KUKA KRL program: MyProgram_219().src

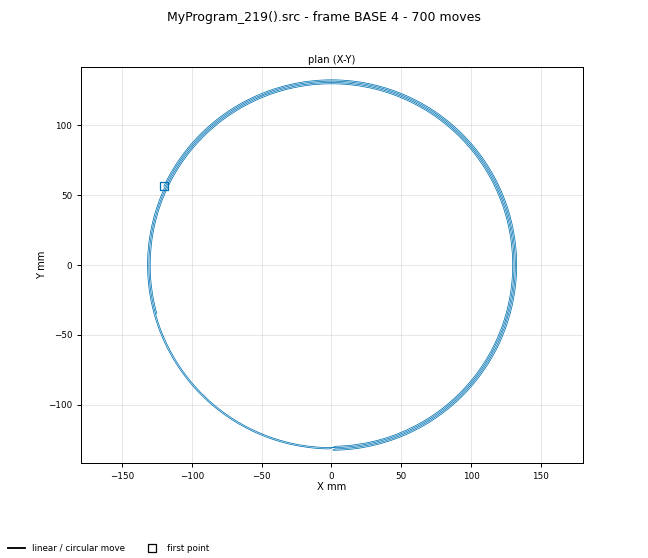
[picture p0: tool path of MyProgram_219().src in frame BASE 4, 700 of 700 moves have a stored position in this frame; points joined in program order, loops and branches not executed]
&ACCESS RVP
&REL 1
&PARAM TEMPLATE = C:\KRC\Roboter\Template\vorgabe
&PARAM EDITMASK = *
DEF MyProgram_219()
; ---- Setting reference (Base) ----
$BASE = BASE_DATA[4]

; --------------------------
; ---- Setting tool (TCP) ----
$TOOL = TOOL_DATA[3]
; --------------------------

$VEL.CP = VEL_APROX_PRINT
Startdeposition()
$VEL.CP = VEL_PRINT
LIN {X -120.0185,Y 56.4143,Z 153,A 151.3812,B 23.2874,C -1.2198,E1 23.1731,E2 655.6773} C_DIS
LIN {X -118.5604,Y 59.4176,Z 153,A 149.9276,B 23.2872,C -1.2236,E1 23.1749,E2 657.1297} C_DIS
LIN {X -117.0207,Y 62.3953,Z 153,A 148.4681,B 23.287,C -1.2274,E1 23.1767,E2 658.5879} C_DIS
LIN {X -115.456,Y 65.2445,Z 153,A 146.9748,B 23.287,C -1.2276,E1 23.1788,E2 660.0893} C_DIS
LIN {X -113.2613,Y 68.9846,Z 153,A 145.0626,B 23.2868,C -1.2313,E1 23.1815,E2 662.0028} C_DIS
LIN {X -110.999,Y 72.5688,Z 153,A 143.3218,B 23.2864,C -1.2405,E1 23.1841,E2 663.7297} C_DIS
LIN {X -108.7297,Y 75.9258,Z 153,A 141.4715,B 23.2864,C -1.2409,E1 23.1871,E2 665.5888} C_DIS
LIN {X -106.1126,Y 79.5432,Z 153,A 139.5664,B 23.286,C -1.2472,E1 23.1902,E2 667.4879} C_DIS
LIN {X -103.5175,Y 82.8922,Z 153,A 137.6938,B 23.2859,C -1.2502,E1 23.1934,E2 669.3624} C_DIS
LIN {X -100.7633,Y 86.2193,Z 153,A 135.8973,B 23.2855,C -1.2582,E1 23.1966,E2 671.1476} C_DIS
LIN {X -98.5031,Y 88.7927,Z 153,A 134.4081,B 23.2853,C -1.2615,E1 23.1994,E2 672.6355} C_DIS
LIN {X -96.2052,Y 91.2772,Z 153,A 132.8552,B 23.2853,C -1.2611,E1 23.2024,E2 674.1968} C_DIS
LIN {X -93.1648,Y 94.3786,Z 153,A 131.0513,B 23.2849,C -1.2689,E1 23.2059,E2 675.9891} C_DIS
LIN {X -90.6941,Y 96.7553,Z 153,A 129.562,B 23.2848,C -1.2721,E1 23.2089,E2 677.4771} C_DIS
LIN {X -88.1572,Y 99.0723,Z 153,A 128.0728,B 23.2846,C -1.2753,E1 23.212,E2 678.9646} C_DIS
LIN {X -85.3531,Y 101.4973,Z 153,A 126.3626,B 23.2846,C -1.274,E1 23.2157,E2 680.6852} C_DIS
LIN {X -82.2555,Y 104.0242,Z 153,A 124.7251,B 23.2843,C -1.2818,E1 23.2192,E2 682.3096} C_DIS
LIN {X -79.5467,Y 106.11,Z 153,A 123.2418,B 23.2841,C -1.2846,E1 23.2225,E2 683.7914} C_DIS
LIN {X -76.3743,Y 108.415,Z 153,A 121.4898,B 23.2841,C -1.2855,E1 23.2265,E2 685.5479} C_DIS
LIN {X -73.2819,Y 110.5295,Z 153,A 119.9361,B 23.2838,C -1.2916,E1 23.2301,E2 687.0917} C_DIS
LIN {X -70.2231,Y 112.497,Z 153,A 118.2317,B 23.2839,C -1.2885,E1 23.2341,E2 688.8097} C_DIS
LIN {X -66.2198,Y 114.8992,Z 153,A 116.2269,B 23.2837,C -1.2927,E1 23.2389,E2 690.8105} C_DIS
LIN {X -62.3991,Y 117.0186,Z 153,A 114.4206,B 23.2833,C -1.2996,E1 23.2433,E2 692.6047} C_DIS
LIN {X -59.4253,Y 118.5564,Z 153,A 112.9705,B 23.2833,C -1.3018,E1 23.2469,E2 694.0535} C_DIS
LIN {X -56.8721,Y 119.7998,Z 153,A 111.7391,B 23.2831,C -1.3036,E1 23.25,E2 695.2838} C_DIS
LIN {X -53.3965,Y 121.3912,Z 153,A 110.0849,B 23.2831,C -1.3059,E1 23.2542,E2 696.9365} C_DIS
LIN {X -50.3517,Y 122.6854,Z 153,A 108.6524,B 23.2829,C -1.3078,E1 23.2579,E2 698.3678} C_DIS
LIN {X -47.2831,Y 123.9004,Z 153,A 107.2236,B 23.2829,C -1.3096,E1 23.2616,E2 699.7954} C_DIS
LIN {X -44.4516,Y 124.9428,Z 153,A 105.9301,B 23.2827,C -1.3117,E1 23.265,E2 701.0862} C_DIS
LIN {X -41.1344,Y 126.0752,Z 153,A 104.4014,B 23.2827,C -1.3128,E1 23.2691,E2 702.6152} C_DIS
LIN {X -38.0368,Y 127.0441,Z 153,A 102.9974,B 23.2826,C -1.3143,E1 23.2728,E2 704.018} C_DIS
LIN {X -34.9435,Y 127.9295,Z 153,A 101.606,B 23.2825,C -1.3157,E1 23.2766,E2 705.4082} C_DIS
LIN {X -31.8497,Y 128.7346,Z 153,A 100.2237,B 23.2825,C -1.317,E1 23.2803,E2 706.7893} C_DIS
LIN {X -28.7581,Y 129.4603,Z 153,A 98.8511,B 23.2824,C -1.3182,E1 23.284,E2 708.1608} C_DIS
LIN {X -26.1134,Y 130.0177,Z 153,A 97.6447,B 23.2824,C -1.3174,E1 23.2873,E2 709.3708} C_DIS
LIN {X -22.593,Y 130.6773,Z 153,A 96.0716,B 23.2824,C -1.3174,E1 23.2917,E2 710.9459} C_DIS
LIN {X -18.9352,Y 131.2551,Z 153,A 94.4964,B 23.2823,C -1.3196,E1 23.296,E2 712.5168} C_DIS
LIN {X -15.475,Y 131.708,Z 153,A 92.9768,B 23.2823,C -1.3199,E1 23.3002,E2 714.0368} C_DIS
LIN {X -11.9161,Y 132.0796,Z 153,A 91.4838,B 23.2821,C -1.3231,E1 23.3043,E2 715.5225} C_DIS
LIN {X -8.9319,Y 132.3147,Z 153,A 90.1919,B 23.2821,C -1.3238,E1 23.3079,E2 716.8134} C_DIS
LIN {X -5.3392,Y 132.5065,Z 153,A 88.5959,B 23.2821,C -1.3223,E1 23.3124,E2 718.4133} C_DIS
LIN {X -1.9248,Y 132.6003,Z 153,A 87.1244,B 23.2821,C -1.3229,E1 23.3165,E2 719.8836} C_DIS
LIN {X 2.9359,Y 132.5835,Z 153,A 84.8957,B 23.2824,C -1.3171,E1 23.3228,E2 722.1267} C_DIS
LIN {X 6.6279,Y 132.4482,Z 153,A 83.4443,B 23.282,C -1.3241,E1 23.3268,E2 723.5601} C_DIS
LIN {X 9.8143,Y 132.2503,Z 153,A 82.0646,B 23.282,C -1.324,E1 23.3306,E2 724.9392} C_DIS
LIN {X 13.086,Y 131.9673,Z 153,A 80.635,B 23.282,C -1.3233,E1 23.3346,E2 726.3697} C_DIS
LIN {X 16.4617,Y 131.5903,Z 153,A 79.1907,B 23.282,C -1.3241,E1 23.3386,E2 727.8108} C_DIS
LIN {X 20.6084,Y 131.0031,Z 153,A 77.3967,B 23.282,C -1.3243,E1 23.3435,E2 729.6025} C_DIS
LIN {X 23.6048,Y 130.4963,Z 153,A 76.0345,B 23.2822,C -1.3215,E1 23.3473,E2 730.9703} C_DIS
LIN {X 26.916,Y 129.8544,Z 153,A 74.5879,B 23.2822,C -1.3213,E1 23.3513,E2 732.4155} C_DIS
LIN {X 30.2955,Y 129.1092,Z 153,A 73.1112,B 23.2822,C -1.3213,E1 23.3553,E2 733.8899} C_DIS
LIN {X 33.027,Y 128.4359,Z 153,A 71.8933,B 23.2822,C -1.3205,E1 23.3586,E2 735.1079} C_DIS
LIN {X 36.4824,Y 127.4991,Z 153,A 70.349,B 23.2822,C -1.3195,E1 23.3627,E2 736.652} C_DIS
LIN {X 39.0613,Y 126.7306,Z 153,A 69.134,B 23.2825,C -1.3161,E1 23.366,E2 737.8732} C_DIS
LIN {X 42.669,Y 125.5642,Z 153,A 67.5494,B 23.2825,C -1.3173,E1 23.3702,E2 739.4515} C_DIS
LIN {X 45.3374,Y 124.6235,Z 153,A 66.2925,B 23.2825,C -1.3145,E1 23.3735,E2 740.7126} C_DIS
LIN {X 48.8073,Y 123.3079,Z 153,A 64.7278,B 23.2825,C -1.3147,E1 23.3776,E2 742.2731} C_DIS
LIN {X 51.3866,Y 122.2532,Z 153,A 63.4941,B 23.2827,C -1.312,E1 23.3807,E2 743.5105} C_DIS
LIN {X 54.6118,Y 120.8476,Z 153,A 61.9862,B 23.2827,C -1.3109,E1 23.3846,E2 745.0173} C_DIS
LIN {X 57.9189,Y 119.2997,Z 153,A 60.4317,B 23.2827,C -1.31,E1 23.3885,E2 746.5696} C_DIS
LIN {X 60.9098,Y 117.8007,Z 153,A 58.9892,B 23.2829,C -1.3083,E1 23.3921,E2 748.0122} C_DIS
LIN {X 63.403,Y 116.477,Z 153,A 57.6835,B 23.2832,C -1.3024,E1 23.3953,E2 749.3287} C_DIS
LIN {X 67.2041,Y 114.3261,Z 153,A 55.8328,B 23.2832,C -1.3014,E1 23.3998,E2 751.1759} C_DIS
LIN {X 70.7142,Y 112.1889,Z 153,A 54.0427,B 23.2834,C -1.2979,E1 23.4041,E2 752.9686} C_DIS
LIN {X 74.3709,Y 109.7989,Z 153,A 52.1811,B 23.2835,C -1.2961,E1 23.4084,E2 754.8281} C_DIS
LIN {X 77.7327,Y 107.4452,Z 153,A 50.3815,B 23.2838,C -1.2917,E1 23.4125,E2 756.632} C_DIS
LIN {X 81.1809,Y 104.8642,Z 153,A 48.5353,B 23.2838,C -1.2891,E1 23.4166,E2 758.4776} C_DIS
LIN {X 84.2506,Y 102.4151,Z 153,A 46.9275,B 23.2838,C -1.2902,E1 23.4201,E2 760.0759} C_DIS
LIN {X 87.0607,Y 100.0365,Z 153,A 45.2407,B 23.2842,C -1.2823,E1 23.4237,E2 761.7756} C_DIS
LIN {X 90.0629,Y 97.3431,Z 153,A 43.608,B 23.2842,C -1.2842,E1 23.427,E2 763.3963} C_DIS
LIN {X 92.9608,Y 94.5787,Z 153,A 41.865,B 23.2844,C -1.2799,E1 23.4305,E2 765.1423} C_DIS
LIN {X 95.7389,Y 91.7656,Z 153,A 40.0792,B 23.2848,C -1.2723,E1 23.434,E2 766.939} C_DIS
LIN {X 98.4971,Y 88.7993,Z 153,A 38.3818,B 23.2848,C -1.2709,E1 23.4372,E2 768.6317} C_DIS
LIN {X 101.3154,Y 85.5698,Z 153,A 36.6033,B 23.2848,C -1.2703,E1 23.4404,E2 770.4031} C_DIS
LIN {X 103.4942,Y 82.9214,Z 153,A 35.136,B 23.285,C -1.2674,E1 23.443,E2 771.8702} C_DIS
LIN {X 105.8539,Y 79.8861,Z 153,A 33.4134,B 23.2854,C -1.2602,E1 23.446,E2 773.602} C_DIS
LIN {X 108.1241,Y 76.7866,Z 153,A 31.8291,B 23.2854,C -1.2598,E1 23.4485,E2 775.1791} C_DIS
LIN {X 110.3638,Y 73.5301,Z 153,A 30.0564,B 23.2858,C -1.2522,E1 23.4513,E2 776.9616} C_DIS
LIN {X 112.7423,Y 69.829,Z 153,A 28.1496,B 23.2861,C -1.2468,E1 23.4542,E2 778.8715} C_DIS
LIN {X 114.9822,Y 66.0764,Z 153,A 26.3687,B 23.2861,C -1.2471,E1 23.4567,E2 780.6416} C_DIS
LIN {X 116.7068,Y 62.9795,Z 153,A 24.731,B 23.2865,C -1.2375,E1 23.4589,E2 782.2942} C_DIS
LIN {X 118.5564,Y 59.4253,Z 153,A 23.1289,B 23.2865,C -1.2392,E1 23.4609,E2 783.8829} C_DIS
LIN {X 120.0148,Y 56.4221,Z 153,A 21.6972,B 23.2866,C -1.2356,E1 23.4626,E2 785.3153} C_DIS
LIN {X 121.2676,Y 53.6728,Z 153,A 20.4109,B 23.2868,C -1.2329,E1 23.4641,E2 786.601} C_DIS
LIN {X 122.5698,Y 50.6284,Z 153,A 18.9867,B 23.287,C -1.229,E1 23.4657,E2 788.0264} C_DIS
LIN {X 123.8752,Y 47.3479,Z 153,A 17.4806,B 23.2871,C -1.2255,E1 23.4672,E2 789.5324} C_DIS
LIN {X 124.8207,Y 44.7903,Z 153,A 16.2864,B 23.2874,C -1.2212,E1 23.4683,E2 790.7302} C_DIS
LIN {X 126.052,Y 41.204,Z 153,A 14.6728,B 23.2875,C -1.2174,E1 23.4698,E2 792.3434} C_DIS
LIN {X 127.0441,Y 38.0368,Z 153,A 13.2519,B 23.2877,C -1.2137,E1 23.4709,E2 793.7648} C_DIS
LIN {X 127.9112,Y 35.009,Z 153,A 11.9126,B 23.2879,C -1.2106,E1 23.4719,E2 795.1035} C_DIS
LIN {X 128.7346,Y 31.8497,Z 153,A 10.5038,B 23.2881,C -1.2063,E1 23.4729,E2 796.5144} C_DIS
LIN {X 129.4603,Y 28.7581,Z 153,A 9.1435,B 23.2883,C -1.2026,E1 23.4738,E2 797.8754} C_DIS
LIN {X 130.1059,Y 25.6797,Z 153,A 7.7968,B 23.2884,C -1.199,E1 23.4745,E2 799.2228} C_DIS
LIN {X 130.5831,Y 23.1195,Z 153,A 6.7047,B 23.2885,C -1.1972,E1 23.4751,E2 800.3126} C_DIS
LIN {X 131.0734,Y 20.1545,Z 153,A 5.3619,B 23.2888,C -1.1908,E1 23.4757,E2 801.663} C_DIS
LIN {X 131.5883,Y 16.4774,Z 153,A 3.8042,B 23.289,C -1.188,E1 23.4762,E2 803.2177} C_DIS
LIN {X 131.9334,Y 13.4374,Z 153,A 2.4944,B 23.2891,C -1.1844,E1 23.4766,E2 804.5282} C_DIS
LIN {X 132.2472,Y 9.8566,Z 153,A 0.9066,B 23.2895,C -1.1776,E1 23.477,E2 806.1228} C_DIS
LIN {X 132.4544,Y 6.5035,Z 153,A -0.5469,B 23.2897,C -1.1728,E1 23.4772,E2 807.5791} C_DIS
LIN {X 132.5999,Y 1.951,Z 153,A -2.4995,B 23.29,C -1.1672,E1 23.4774,E2 809.5332} C_DIS
LIN {X 132.6105,Y -0.9415,Z 153,A -3.7215,B 23.29,C -1.1645,E1 23.4774,E2 810.7539} C_DIS
LIN {X 132.5171,Y -5.0689,Z 153,A -5.4928,B 23.2903,C -1.1594,E1 23.4772,E2 812.5269} C_DIS
LIN {X 132.3401,Y -8.5247,Z 153,A -6.9651,B 23.2905,C -1.1557,E1 23.477,E2 813.999} C_DIS
LIN {X 132.0802,Y -11.9083,Z 153,A -8.3941,B 23.2906,C -1.1528,E1 23.4766,E2 815.4262} C_DIS
LIN {X 131.6676,Y -15.8141,Z 153,A -10.1033,B 23.2909,C -1.1466,E1 23.4761,E2 817.1398} C_DIS
LIN {X 131.2563,Y -18.9271,Z 153,A -11.466,B 23.2911,C -1.1419,E1 23.4756,E2 818.5057} C_DIS
LIN {X 130.6787,Y -22.5851,Z 153,A -13.0213,B 23.2913,C -1.139,E1 23.4749,E2 820.0585} C_DIS
LIN {X 130.1811,Y -25.2871,Z 153,A -14.2322,B 23.2915,C -1.134,E1 23.4742,E2 821.2744} C_DIS
LIN {X 129.4621,Y -28.7502,Z 153,A -15.7214,B 23.2917,C -1.131,E1 23.4734,E2 822.7616} C_DIS
LIN {X 128.5056,Y -32.7522,Z 153,A -17.5015,B 23.2919,C -1.1252,E1 23.4722,E2 824.5451} C_DIS
LIN {X 127.6253,Y -36.0315,Z 153,A -18.9893,B 23.2922,C -1.1195,E1 23.4711,E2 826.0382} C_DIS
LIN {X 126.5736,Y -39.5742,Z 153,A -20.5353,B 23.2922,C -1.117,E1 23.4698,E2 827.5809} C_DIS
LIN {X 125.6993,Y -42.2632,Z 153,A -21.7708,B 23.2925,C -1.1124,E1 23.4687,E2 828.8203} C_DIS
LIN {X 124.4755,Y -45.7477,Z 153,A -23.3361,B 23.2927,C -1.109,E1 23.4673,E2 830.3848} C_DIS
LIN {X 123.3079,Y -48.8073,Z 153,A -24.741,B 23.2928,C -1.1051,E1 23.4659,E2 831.791} C_DIS
LIN {X 122.2841,Y -51.3126,Z 153,A -25.9212,B 23.293,C -1.101,E1 23.4646,E2 832.9745} C_DIS
LIN {X 120.9147,Y -54.4616,Z 153,A -27.371,B 23.2931,C -1.0981,E1 23.463,E2 834.4229} C_DIS
LIN {X 119.5106,Y -57.4773,Z 153,A -28.828,B 23.2934,C -1.0928,E1 23.4612,E2 835.8849} C_DIS
LIN {X 117.8007,Y -60.9098,Z 153,A -30.4567,B 23.2935,C -1.0892,E1 23.4592,E2 837.5132} C_DIS
LIN {X 116.3772,Y -63.586,Z 153,A -31.8054,B 23.2938,C -1.0833,E1 23.4574,E2 838.8689} C_DIS
LIN {X 114.2709,Y -67.298,Z 153,A -33.6824,B 23.2941,C -1.0763,E1 23.4547,E2 840.7533} C_DIS
LIN {X 111.921,Y -71.1386,Z 153,A -35.5264,B 23.2941,C -1.0758,E1 23.452,E2 842.5883} C_DIS
LIN {X 109.8274,Y -74.3288,Z 153,A -37.232,B 23.2944,C -1.0683,E1 23.4494,E2 844.3037} C_DIS
LIN {X 107.6309,Y -77.4765,Z 153,A -38.8145,B 23.2944,C -1.0675,E1 23.4468,E2 845.8797} C_DIS
LIN {X 105.5981,Y -80.225,Z 153,A -40.2823,B 23.2946,C -1.064,E1 23.4444,E2 847.3489} C_DIS
LIN {X 103.4942,Y -82.9214,Z 153,A -41.835,B 23.295,C -1.0562,E1 23.4416,E2 848.9134} C_DIS
LIN {X 100.7633,Y -86.2193,Z 153,A -43.5915,B 23.295,C -1.0561,E1 23.4385,E2 850.6615} C_DIS
LIN {X 98.5031,Y -88.7927,Z 153,A -45.0636,B 23.2951,C -1.0527,E1 23.4358,E2 852.135} C_DIS
LIN {X 96.1695,Y -91.315,Z 153,A -46.5193,B 23.2952,C -1.0504,E1 23.433,E2 853.5895} C_DIS
LIN {X 93.7768,Y -93.7705,Z 153,A -48.1152,B 23.2956,C -1.0409,E1 23.4298,E2 855.202} C_DIS
LIN {X 90.6941,Y -96.7553,Z 153,A -49.8566,B 23.2956,C -1.0422,E1 23.4263,E2 856.9323} C_DIS
LIN {X 88.1572,Y -99.0723,Z 153,A -51.3324,B 23.2956,C -1.0391,E1 23.4233,E2 858.4094} C_DIS
LIN {X 85.5698,Y -101.3154,Z 153,A -52.7981,B 23.2958,C -1.0364,E1 23.4202,E2 859.8757} C_DIS
LIN {X 82.6822,Y -103.6846,Z 153,A -54.5007,B 23.2961,C -1.0284,E1 23.4164,E2 861.5916} C_DIS
LIN {X 79.0894,Y -106.4505,Z 153,A -56.3994,B 23.2961,C -1.0272,E1 23.4122,E2 863.4857} C_DIS
LIN {X 75.5577,Y -108.9858,Z 153,A -58.3154,B 23.2964,C -1.0215,E1 23.4078,E2 865.4091} C_DIS
LIN {X 71.8604,Y -111.4589,Z 153,A -60.14,B 23.2964,C -1.0226,E1 23.4036,E2 867.2244} C_DIS
LIN {X 68.9846,Y -113.2613,Z 153,A -61.5988,B 23.2964,C -1.0202,E1 23.4001,E2 868.6843} C_DIS
LIN {X 66.0764,Y -114.9822,Z 153,A -63.0515,B 23.2966,C -1.0179,E1 23.3966,E2 870.1379} C_DIS
LIN {X 62.8825,Y -116.7589,Z 153,A -64.7151,B 23.2969,C -1.0109,E1 23.3925,E2 871.8139} C_DIS
LIN {X 59.4253,Y -118.5564,Z 153,A -66.2983,B 23.2968,C -1.0131,E1 23.3886,E2 873.3869} C_DIS
LIN {X 56.9163,Y -119.7787,Z 153,A -67.494,B 23.2968,C -1.0117,E1 23.3856,E2 874.5827} C_DIS
LIN {X 53.8486,Y -121.1889,Z 153,A -68.9478,B 23.2969,C -1.0097,E1 23.3819,E2 876.0377} C_DIS
LIN {X 50.6868,Y -122.5454,Z 153,A -70.4194,B 23.2969,C -1.0082,E1 23.3781,E2 877.5092} C_DIS
LIN {X 47.2831,Y -123.9004,Z 153,A -72.0079,B 23.2971,C -1.0057,E1 23.374,E2 879.1002} C_DIS
LIN {X 44.707,Y -124.8507,Z 153,A -73.2383,B 23.2972,C -1.002,E1 23.3707,E2 880.3372} C_DIS
LIN {X 41.1344,Y -126.0752,Z 153,A -74.8143,B 23.2972,C -1.0027,E1 23.3666,E2 881.9081} C_DIS
LIN {X 38.0368,Y -127.0441,Z 153,A -76.211,B 23.2972,C -1.0014,E1 23.3628,E2 883.3056} C_DIS
LIN {X 34.9435,Y -127.9295,Z 153,A -77.5957,B 23.2973,C -1.0001,E1 23.3591,E2 884.6909} C_DIS
LIN {X 32.039,Y -128.6866,Z 153,A -78.8599,B 23.2973,C -1.0004,E1 23.3557,E2 885.9522} C_DIS
LIN {X 29.315,Y -129.3331,Z 153,A -80.1109,B 23.2974,C -0.9972,E1 23.3523,E2 887.2094} C_DIS
LIN {X 25.6797,Y -130.1059,Z 153,A -81.6928,B 23.2974,C -0.997,E1 23.348,E2 888.7898} C_DIS
LIN {X 22.9082,Y -130.6209,Z 153,A -82.9272,B 23.2975,C -0.9952,E1 23.3446,E2 890.0272} C_DIS
LIN {X 18.9609,Y -131.2514,Z 153,A -84.6446,B 23.2975,C -0.9945,E1 23.3398,E2 891.7447} C_DIS
LIN {X 15.7554,Y -131.6746,Z 153,A -86.0399,B 23.2975,C -0.9937,E1 23.336,E2 893.1408} C_DIS
LIN {X 12.4799,Y -132.0255,Z 153,A -87.4629,B 23.2975,C -0.9929,E1 23.332,E2 894.5647} C_DIS
LIN {X 8.9114,Y -132.3162,Z 153,A -88.9797,B 23.2975,C -0.9937,E1 23.3278,E2 896.0789} C_DIS
LIN {X 3.8989,Y -132.5568,Z 153,A -91.2084,B 23.2977,C -0.99,E1 23.3215,E2 898.3162} C_DIS
LIN {X 0.9369,Y -132.6077,Z 153,A -92.0457,B 23.2969,C -1.0112,E1 23.3194,E2 899.0997} C_DIS
Enddeposition()
LIN {X 0.9369,Y -132.6077,Z 153,A -92.0457,B 23.2969,C -1.0112,E1 23.3194,E2 899.0997} C_DIS
Startdeposition()
$VEL.CP = VEL_PRINT
LIN {X 2.3502,Y -131.6529,Z 153,A -90.8514,B 22.2978,C -0.8695,E1 22.3183,E2 898.1516} C_DIS
LIN {X 6.558,Y -131.5103,Z 153,A -89.0359,B 22.2978,C -0.8694,E1 22.3233,E2 896.337} C_DIS
LIN {X 10.8155,Y -131.229,Z 153,A -87.1803,B 22.2978,C -0.8702,E1 22.3285,E2 894.4805} C_DIS
LIN {X 14.3146,Y -130.8934,Z 153,A -85.6847,B 22.2978,C -0.8694,E1 22.3326,E2 892.9879} C_DIS
LIN {X 18.2026,Y -130.4101,Z 153,A -83.7965,B 22.2974,C -0.8791,E1 22.3379,E2 891.076} C_DIS
LIN {X 22.0211,Y -129.8196,Z 153,A -82.2316,B 22.2976,C -0.8748,E1 22.3422,E2 889.5241} C_DIS
LIN {X 27.5629,Y -128.7565,Z 153,A -80.0882,B 22.298,C -0.8621,E1 22.348,E2 887.4171} C_DIS
LIN {X 29.4629,Y -128.335,Z 153,A -79.0109,B 22.2976,C -0.8738,E1 22.351,E2 886.3108} C_DIS
LIN {X 33.0947,Y -127.4487,Z 153,A -77.3837,B 22.2976,C -0.8754,E1 22.3554,E2 884.6822} C_DIS
LIN {X 38.7328,Y -125.8479,Z 153,A -74.7637,B 22.2973,C -0.8815,E1 22.3625,E2 882.0511} C_DIS
LIN {X 42.1515,Y -124.7456,Z 153,A -73.3003,B 22.2974,C -0.8787,E1 22.3663,E2 880.5985} C_DIS
LIN {X 45.6252,Y -123.5174,Z 153,A -71.4667,B 22.2969,C -0.8918,E1 22.3712,E2 878.7347} C_DIS
LIN {X 49.9299,Y -121.8418,Z 153,A -69.6991,B 22.2973,C -0.8829,E1 22.3757,E2 876.9949} C_DIS
LIN {X 52.3421,Y -120.8228,Z 153,A -68.5334,B 22.2972,C -0.8859,E1 22.3787,E2 875.8246} C_DIS
LIN {X 55.6372,Y -119.342,Z 153,A -66.9756,B 22.2971,C -0.8876,E1 22.3827,E2 874.2667} C_DIS
LIN {X 59.9235,Y -117.2478,Z 153,A -64.8252,B 22.2968,C -0.8945,E1 22.3881,E2 872.1047} C_DIS
LIN {X 63.7063,Y -115.2383,Z 153,A -62.9608,B 22.2968,C -0.8977,E1 22.3927,E2 870.2379} C_DIS
LIN {X 67.6763,Y -112.9529,Z 153,A -60.9935,B 22.2966,C -0.9001,E1 22.3974,E2 868.2713} C_DIS
LIN {X 71.1485,Y -110.7983,Z 153,A -59.2373,B 22.2966,C -0.9024,E1 22.4015,E2 866.5155} C_DIS
LIN {X 74.7504,Y -108.4012,Z 153,A -57.3386,B 22.2964,C -0.9069,E1 22.4059,E2 864.6123} C_DIS
LIN {X 79.4099,Y -105.0353,Z 153,A -54.2763,B 22.2951,C -0.9396,E1 22.413,E2 861.4767} C_DIS
LIN {X 83.4138,Y -101.8847,Z 153,A -52.9808,B 22.2966,C -0.8994,E1 22.4155,E2 860.2922} C_DIS
LIN {X 87.8516,Y -98.0838,Z 153,A -50.2415,B 22.2961,C -0.9146,E1 22.4214,E2 857.5249} C_DIS
LIN {X 90.3601,Y -95.7778,Z 153,A -48.6324,B 22.2957,C -0.9243,E1 22.4247,E2 855.8981} C_DIS
LIN {X 93.5629,Y -92.6519,Z 153,A -46.0905,B 22.2943,C -0.9583,E1 22.4299,E2 853.2793} C_DIS
LIN {X 97.2341,Y -88.7922,Z 153,A -44.2689,B 22.2951,C -0.9396,E1 22.4332,E2 851.5159} C_DIS
LIN {X 101.5927,Y -83.7695,Z 153,A -41.6245,B 22.2953,C -0.9348,E1 22.438,E2 848.8977} C_DIS
LIN {X 105.3967,Y -78.9303,Z 153,A -38.8961,B 22.2949,C -0.9444,E1 22.4426,E2 846.1587} C_DIS
LIN {X 107.8084,Y -75.603,Z 153,A -37.0332,B 22.2945,C -0.9529,E1 22.4457,E2 844.2837} C_DIS
LIN {X 110.3428,Y -71.8529,Z 153,A -35.1217,B 22.2945,C -0.9556,E1 22.4486,E2 842.3761} C_DIS
LIN {X 112.5666,Y -68.3166,Z 153,A -33.3083,B 22.2942,C -0.9605,E1 22.4513,E2 840.5602} C_DIS
LIN {X 114.7715,Y -64.5435,Z 153,A -31.421,B 22.294,C -0.9653,E1 22.4539,E2 838.6713} C_DIS
LIN {X 117.6,Y -59.2318,Z 153,A -28.925,B 22.294,C -0.967,E1 22.4571,E2 836.186} C_DIS
LIN {X 118.8969,Y -56.5809,Z 153,A -27.6252,B 22.2938,C -0.9716,E1 22.4587,E2 834.882} C_DIS
LIN {X 120.5658,Y -52.9365,Z 153,A -25.7876,B 22.2934,C -0.9815,E1 22.4608,E2 833.0299} C_DIS
LIN {X 122.759,Y -47.6244,Z 153,A -23.61,B 22.2937,C -0.9732,E1 22.4631,E2 830.8878} C_DIS
LIN {X 123.5789,Y -45.461,Z 153,A -22.4444,B 22.2932,C -0.9841,E1 22.4642,E2 829.701} C_DIS
LIN {X 124.5714,Y -42.6624,Z 153,A -21.0174,B 22.2928,C -0.9948,E1 22.4655,E2 828.2549} C_DIS
LIN {X 127.5962,Y -32.5132,Z 153,A -16.8433,B 22.2931,C -0.9877,E1 22.4688,E2 824.1266} C_DIS
LIN {X 128.6682,Y -27.9722,Z 153,A -14.8033,B 22.2928,C -0.9946,E1 22.4701,E2 822.082} C_DIS
LIN {X 129.1788,Y -25.5207,Z 153,A -13.3709,B 22.2919,C -1.015,E1 22.4709,E2 820.6057} C_DIS
LIN {X 129.9745,Y -21.0929,Z 153,A -11.5859,B 22.292,C -1.0127,E1 22.4717,E2 818.8385} C_DIS
LIN {X 130.3573,Y -18.5716,Z 153,A -10.4416,B 22.2918,C -1.018,E1 22.4722,E2 817.688} C_DIS
LIN {X 130.8402,Y -14.8056,Z 153,A -8.7225,B 22.2914,C -1.0266,E1 22.4728,E2 815.9578} C_DIS
LIN {X 131.148,Y -11.7744,Z 153,A -7.5271,B 22.2915,C -1.0244,E1 22.4731,E2 814.7762} C_DIS
LIN {X 131.3444,Y -9.3107,Z 153,A -6.4382,B 22.2913,C -1.0286,E1 22.4733,E2 813.6837} C_DIS
LIN {X 131.5505,Y -5.7275,Z 153,A -4.7498,B 22.2908,C -1.0399,E1 22.4735,E2 811.9772} C_DIS
LIN {X 131.6627,Y -1.7621,Z 153,A -3.0226,B 22.2906,C -1.0455,E1 22.4736,E2 810.2469} C_DIS
LIN {X 131.6661,Y 1.5596,Z 153,A -1.7216,B 22.2907,C -1.043,E1 22.4736,E2 808.9613} C_DIS
LIN {X 131.5584,Y 5.5239,Z 153,A 0.1236,B 22.2902,C -1.0545,E1 22.4734,E2 807.0985} C_DIS
LIN {X 131.3217,Y 9.6215,Z 153,A 1.8019,B 22.2902,C -1.0548,E1 22.4731,E2 805.4305} C_DIS
LIN {X 130.9317,Y 13.9588,Z 153,A 3.7387,B 22.2898,C -1.063,E1 22.4726,E2 803.4854} C_DIS
LIN {X 130.5388,Y 17.2506,Z 153,A 5.1182,B 22.2898,C -1.0644,E1 22.4721,E2 802.1115} C_DIS
LIN {X 130.0964,Y 20.3194,Z 153,A 6.4488,B 22.2896,C -1.0677,E1 22.4716,E2 800.781} C_DIS
LIN {X 129.4087,Y 24.3201,Z 153,A 8.4061,B 22.2889,C -1.0827,E1 22.4706,E2 798.7975} C_DIS
LIN {X 127.8056,Y 31.6846,Z 153,A 11.6321,B 22.2886,C -1.0902,E1 22.4686,E2 795.5731} C_DIS
LIN {X 126.9858,Y 34.8273,Z 153,A 13.0165,B 22.2884,C -1.093,E1 22.4676,E2 794.1903} C_DIS
LIN {X 125.6715,Y 39.3087,Z 153,A 14.8473,B 22.2886,C -1.0893,E1 22.4661,E2 792.3813} C_DIS
LIN {X 124.4068,Y 43.1372,Z 153,A 16.6306,B 22.2883,C -1.096,E1 22.4645,E2 790.5918} C_DIS
LIN {X 123.1684,Y 46.557,Z 153,A 18.1842,B 22.2881,C -1.0992,E1 22.463,E2 789.0396} C_DIS
LIN {X 121.9264,Y 49.7202,Z 153,A 19.5984,B 22.2881,C -1.1003,E1 22.4615,E2 787.6312} C_DIS
LIN {X 120.7711,Y 52.4618,Z 153,A 20.9067,B 22.2879,C -1.1048,E1 22.4601,E2 786.3195} C_DIS
LIN {X 118.5538,Y 57.2976,Z 153,A 23.2127,B 22.2876,C -1.1109,E1 22.4574,E2 784.0116} C_DIS
LIN {X 117.1002,Y 60.2135,Z 153,A 24.6312,B 22.2874,C -1.1149,E1 22.4556,E2 782.5912} C_DIS
LIN {X 115.3888,Y 63.4345,Z 153,A 26.3428,B 22.2869,C -1.1253,E1 22.4533,E2 780.8626} C_DIS
LIN {X 113.0177,Y 67.5675,Z 153,A 28.3245,B 22.2869,C -1.1264,E1 22.4505,E2 778.8896} C_DIS
LIN {X 110.8121,Y 71.1271,Z 153,A 30.1689,B 22.2866,C -1.1322,E1 22.4477,E2 777.0404} C_DIS
LIN {X 108.3662,Y 74.8013,Z 153,A 32.1095,B 22.2863,C -1.1381,E1 22.4447,E2 775.0952} C_DIS
LIN {X 105.8817,Y 78.2787,Z 153,A 33.9736,B 22.286,C -1.143,E1 22.4416,E2 773.2287} C_DIS
LIN {X 103.174,Y 81.8139,Z 153,A 36.2992,B 22.2849,C -1.1666,E1 22.4375,E2 770.8536} C_DIS
LIN {X 100.3887,Y 85.2082,Z 153,A 37.5985,B 22.2861,C -1.1414,E1 22.4353,E2 769.6271} C_DIS
LIN {X 97.955,Y 87.9955,Z 153,A 39.3104,B 22.2857,C -1.15,E1 22.4321,E2 767.9014} C_DIS
LIN {X 95.1444,Y 91.0268,Z 153,A 41.1536,B 22.2854,C -1.1561,E1 22.4286,E2 766.0512} C_DIS
LIN {X 91.9917,Y 94.2123,Z 153,A 43.8288,B 22.2834,C -1.1953,E1 22.4231,E2 763.2857} C_DIS
LIN {X 87.6436,Y 98.27,Z 153,A 45.5173,B 22.2854,C -1.1572,E1 22.4198,E2 761.7052} C_DIS
LIN {X 84.3341,Y 101.125,Z 153,A 47.5235,B 22.2849,C -1.1658,E1 22.4155,E2 759.6851} C_DIS
LIN {X 81.2519,Y 103.617,Z 153,A 49.2363,B 22.2848,C -1.1685,E1 22.4117,E2 757.9726} C_DIS
LIN {X 77.8086,Y 106.2271,Z 153,A 51.1574,B 22.2845,C -1.1738,E1 22.4074,E2 756.0454} C_DIS
LIN {X 74.0939,Y 108.8511,Z 153,A 53.1574,B 22.2843,C -1.1781,E1 22.4028,E2 754.0418} C_DIS
LIN {X 70.4749,Y 111.2281,Z 153,A 55.0185,B 22.2843,C -1.1801,E1 22.3985,E2 752.1825} C_DIS
LIN {X 66.7257,Y 113.5166,Z 153,A 57.0024,B 22.2839,C -1.1864,E1 22.3937,E2 750.1891} C_DIS
LIN {X 62.597,Y 115.845,Z 153,A 59.0098,B 22.2839,C -1.1866,E1 22.3888,E2 748.1876} C_DIS
LIN {X 57.8296,Y 118.2954,Z 153,A 61.1796,B 22.2841,C -1.182,E1 22.3834,E2 746.0367} C_DIS
LIN {X 54.9361,Y 119.6662,Z 153,A 62.5583,B 22.2841,C -1.183,E1 22.3799,E2 744.6593} C_DIS
LIN {X 51.8853,Y 121.0203,Z 153,A 64.0595,B 22.2839,C -1.1869,E1 22.3761,E2 743.1519} C_DIS
LIN {X 47.4119,Y 122.8416,Z 153,A 66.0037,B 22.2841,C -1.1818,E1 22.3711,E2 741.2263} C_DIS
LIN {X 44.5076,Y 123.9232,Z 153,A 67.4763,B 22.2838,C -1.1888,E1 22.3672,E2 739.7387} C_DIS
LIN {X 40.941,Y 125.1487,Z 153,A 69.0967,B 22.2838,C -1.1892,E1 22.3629,E2 738.1208} C_DIS
LIN {X 37.8299,Y 126.1242,Z 153,A 70.9523,B 22.2827,C -1.2107,E1 22.3578,E2 736.2125} C_DIS
LIN {X 34.2335,Y 127.1458,Z 153,A 72.1168,B 22.2837,C -1.1903,E1 22.3548,E2 735.1037} C_DIS
LIN {X 30.6891,Y 128.0473,Z 153,A 73.7381,B 22.2836,C -1.1926,E1 22.3504,E2 733.4789} C_DIS
LIN {X 27.0498,Y 128.8673,Z 153,A 75.5263,B 22.2831,C -1.2011,E1 22.3455,E2 731.6713} C_DIS
LIN {X 23.2162,Y 129.6107,Z 153,A 77.0767,B 22.2835,C -1.1949,E1 22.3413,E2 730.139} C_DIS
LIN {X 19.5247,Y 130.2195,Z 153,A 78.9238,B 22.2829,C -1.2055,E1 22.3361,E2 728.2659} C_DIS
LIN {X 14.5738,Y 130.8655,Z 153,A 80.8522,B 22.2835,C -1.1948,E1 22.3308,E2 726.3676} C_DIS
LIN {X 11.2594,Y 131.1915,Z 153,A 82.3089,B 22.2835,C -1.1953,E1 22.3268,E2 724.9103} C_DIS
LIN {X 7.9105,Y 131.436,Z 153,A 83.7819,B 22.2835,C -1.196,E1 22.3227,E2 723.4366} C_DIS
LIN {X 3.4253,Y 131.6294,Z 153,A 85.6873,B 22.2835,C -1.1937,E1 22.3174,E2 721.5378} C_DIS
LIN {X -0.0037,Y 131.6758,Z 153,A 87.2081,B 22.2835,C -1.1947,E1 22.3131,E2 720.0144} C_DIS
LIN {X -3.5557,Y 131.6258,Z 153,A 88.7916,B 22.2835,C -1.1961,E1 22.3087,E2 718.4271} C_DIS
LIN {X -7.328,Y 131.4716,Z 153,A 90.5806,B 22.2831,C -1.2021,E1 22.3037,E2 716.6216} C_DIS
LIN {X -11.2579,Y 131.1916,Z 153,A 92.311,B 22.2831,C -1.2021,E1 22.2988,E2 714.8902} C_DIS
LIN {X -14.9193,Y 130.8275,Z 153,A 93.6669,B 22.2837,C -1.1903,E1 22.2952,E2 713.5648} C_DIS
LIN {X -17.5906,Y 130.4942,Z 153,A 94.9829,B 22.2834,C -1.1961,E1 22.2915,E2 712.2323} C_DIS
LIN {X -21.5882,Y 129.8918,Z 153,A 97.0852,B 22.2827,C -1.2103,E1 22.2856,E2 710.0902} C_DIS
LIN {X -25.5138,Y 129.1802,Z 153,A 98.3695,B 22.2838,C -1.1887,E1 22.2822,E2 708.8615} C_DIS
LIN {X -30.1241,Y 128.1828,Z 153,A 100.9139,B 22.2827,C -1.2089,E1 22.2751,E2 706.2599} C_DIS
LIN {X -33.9236,Y 127.2284,Z 153,A 102.1908,B 22.2838,C -1.1881,E1 22.2718,E2 705.0358} C_DIS
LIN {X -37.7433,Y 126.1504,Z 153,A 104.074,B 22.2835,C -1.1932,E1 22.2667,E2 703.1356} C_DIS
LIN {X -41.7398,Y 124.8827,Z 153,A 105.7299,B 22.284,C -1.1837,E1 22.2624,E2 701.5015} C_DIS
LIN {X -45.1569,Y 123.6891,Z 153,A 107.4207,B 22.2839,C -1.1868,E1 22.2579,E2 699.7986} C_DIS
LIN {X -54.8465,Y 119.7076,Z 153,A 111.7348,B 22.2847,C -1.1696,E1 22.2469,E2 695.519} C_DIS
LIN {X -56.9873,Y 118.7028,Z 153,A 113.007,B 22.2843,C -1.1787,E1 22.2436,E2 694.219} C_DIS
LIN {X -60.4326,Y 116.9886,Z 153,A 114.5922,B 22.2846,C -1.172,E1 22.2397,E2 692.6466} C_DIS
LIN {X -63.7896,Y 115.1922,Z 153,A 116.3535,B 22.2846,C -1.1738,E1 22.2353,E2 690.8748} C_DIS
LIN {X -67.4466,Y 113.0898,Z 153,A 118.1824,B 22.2847,C -1.1703,E1 22.2309,E2 689.0491} C_DIS
LIN {X -71.2321,Y 110.7448,Z 153,A 120.2599,B 22.2846,C -1.1728,E1 22.226,E2 686.9574} C_DIS
LIN {X -75.0985,Y 108.1599,Z 153,A 122.1586,B 22.285,C -1.1634,E1 22.2217,E2 685.0764} C_DIS
LIN {X -78.5662,Y 105.6679,Z 153,A 124.0156,B 22.2852,C -1.1595,E1 22.2175,E2 683.2221} C_DIS
LIN {X -81.8238,Y 103.1662,Z 153,A 125.852,B 22.2853,C -1.1579,E1 22.2134,E2 681.3824} C_DIS
LIN {X -85.2558,Y 100.3484,Z 153,A 127.7765,B 22.2855,C -1.1533,E1 22.2093,E2 679.4616} C_DIS
LIN {X -88.5491,Y 97.4546,Z 153,A 129.6675,B 22.2858,C -1.1483,E1 22.2054,E2 677.5754} C_DIS
LIN {X -91.5583,Y 94.6331,Z 153,A 131.4646,B 22.286,C -1.1442,E1 22.2018,E2 675.7807} C_DIS
LIN {X -94.4959,Y 91.7001,Z 153,A 133.3369,B 22.286,C -1.1427,E1 22.1981,E2 673.9033} C_DIS
LIN {X -97.5952,Y 88.3942,Z 153,A 135.2744,B 22.2864,C -1.1363,E1 22.1944,E2 671.9731} C_DIS
LIN {X -100.3146,Y 85.2955,Z 153,A 137.088,B 22.2866,C -1.1326,E1 22.1911,E2 670.16} C_DIS
LIN {X -103.1007,Y 81.9061,Z 153,A 139.027,B 22.2867,C -1.1289,E1 22.1877,E2 668.2205} C_DIS
LIN {X -105.8347,Y 78.3422,Z 153,A 141.0148,B 22.2869,C -1.1251,E1 22.1844,E2 666.2319} C_DIS
LIN {X -108.3636,Y 74.8052,Z 153,A 142.9173,B 22.2871,C -1.1204,E1 22.1813,E2 664.3313} C_DIS
LIN {X -111.1245,Y 70.6389,Z 153,A 145.0506,B 22.2875,C -1.1125,E1 22.1781,E2 662.2066} C_DIS
LIN {X -113.2117,Y 67.2422,Z 153,A 146.8202,B 22.2877,C -1.1091,E1 22.1755,E2 660.4357} C_DIS
LIN {X -115.4045,Y 63.4059,Z 153,A 148.7181,B 22.288,C -1.1025,E1 22.173,E2 658.5441} C_DIS
LIN {X -116.8091,Y 60.7759,Z 153,A 150.0196,B 22.2882,C -1.0989,E1 22.1713,E2 657.2442} C_DIS
LIN {X -118.5039,Y 57.4035,Z 153,A 151.6788,B 22.2883,C -1.0947,E1 22.1692,E2 655.5859} C_DIS
LIN {X -119.6908,Y 54.8829,Z 153,A 152.8357,B 22.2886,C -1.0888,E1 22.1679,E2 654.4376} C_DIS
LIN {X -120.995,Y 51.944,Z 153,A 154.2661,B 22.2888,C -1.0859,E1 22.1663,E2 653.0059} C_DIS
LIN {X -122.3471,Y 48.6763,Z 153,A 155.7877,B 22.289,C -1.0804,E1 22.1647,E2 651.489} C_DIS
LIN {X -123.6011,Y 45.4007,Z 153,A 157.4967,B 22.2889,C -1.0835,E1 22.163,E2 649.761} C_DIS
LIN {X -124.9965,Y 41.398,Z 153,A 159.1425,B 22.2895,C -1.0694,E1 22.1615,E2 648.1419} C_DIS
LIN {X -125.7813,Y 38.9502,Z 153,A 160.2116,B 22.2898,C -1.0638,E1 22.1606,E2 647.0806} C_DIS
LIN {X -126.5259,Y 36.4608,Z 153,A 161.459,B 22.2898,C -1.0652,E1 22.1597,E2 645.8214} C_DIS
LIN {X -127.2253,Y 33.9354,Z 153,A 162.636,B 22.2898,C -1.0632,E1 22.1588,E2 644.6419} C_DIS
LIN {X -128.0509,Y 30.674,Z 153,A 164.1217,B 22.29,C -1.0595,E1 22.1578,E2 643.1562} C_DIS
LIN {X -128.7461,Y 27.6114,Z 153,A 165.5136,B 22.2901,C -1.0562,E1 22.157,E2 641.7637} C_DIS
LIN {X -129.5838,Y 23.3664,Z 153,A 167.3562,B 22.2905,C -1.0485,E1 22.156,E2 639.9291} C_DIS
LIN {X -130.1206,Y 20.1631,Z 153,A 168.8073,B 22.2905,C -1.0456,E1 22.1554,E2 638.476} C_DIS
LIN {X -130.6433,Y 16.4534,Z 153,A 170.9922,B 22.2898,C -1.0639,E1 22.1546,E2 636.2275} C_DIS
LIN {X -131.124,Y 12.0315,Z 153,A 172.3481,B 22.2911,C -1.033,E1 22.1542,E2 634.9443} C_DIS
LIN {X -131.4056,Y 8.4041,Z 153,A 174.032,B 22.2911,C -1.0322,E1 22.1539,E2 633.2511} C_DIS
LIN {X -131.587,Y 4.7911,Z 153,A 176.1293,B 22.2904,C -1.0494,E1 22.1537,E2 631.0938} C_DIS
LIN {X -131.6735,Y 0.312,Z 153,A 177.4654,B 22.2918,C -1.0171,E1 22.1537,E2 629.8345} C_DIS
LIN {X -131.488,Y -7.0019,Z 153,A -179.2967,B 22.2922,C -1.0091,E1 22.1539,E2 626.5955} C_DIS
LIN {X -130.9785,Y -13.524,Z 153,A -176.4892,B 22.2926,C -0.9983,E1 22.1546,E2 623.7975} C_DIS
LIN {X -130.2939,Y -19.0158,Z 153,A -174.134,B 22.2931,C -0.9884,E1 22.1554,E2 621.4525} C_DIS
LIN {X -129.8882,Y -21.6098,Z 153,A -172.8016,B 22.2929,C -0.9929,E1 22.156,E2 620.0993} C_DIS
LIN {X -129.3126,Y -24.8231,Z 153,A -171.3172,B 22.2929,C -0.9912,E1 22.1568,E2 618.6094} C_DIS
LIN {X -128.613,Y -28.2276,Z 153,A -169.9017,B 22.2933,C -0.9823,E1 22.1576,E2 617.2078} C_DIS
LIN {X -128.0413,Y -30.7139,Z 153,A -168.7352,B 22.2933,C -0.9813,E1 22.1583,E2 616.0362} C_DIS
LIN {X -127.2309,Y -33.9142,Z 153,A -167.2971,B 22.2935,C -0.977,E1 22.1593,E2 614.6001} C_DIS
LIN {X -126.3558,Y -37.0418,Z 153,A -165.8467,B 22.2937,C -0.9743,E1 22.1605,E2 613.1472} C_DIS
LIN {X -125.3392,Y -40.349,Z 153,A -164.3711,B 22.2939,C -0.9685,E1 22.1617,E2 611.6774} C_DIS
LIN {X -123.2833,Y -46.2503,Z 153,A -160.9601,B 22.293,C -0.9902,E1 22.165,E2 608.1868} C_DIS
LIN {X -121.443,Y -50.8867,Z 153,A -159.1033,B 22.2938,C -0.9704,E1 22.167,E2 606.371} C_DIS
LIN {X -120.1287,Y -53.9163,Z 153,A -157.8907,B 22.2944,C -0.9566,E1 22.1683,E2 605.1874} C_DIS
LIN {X -118.6068,Y -57.1881,Z 153,A -156.4263,B 22.2947,C -0.9476,E1 22.17,E2 603.7377} C_DIS
LIN {X -117.2152,Y -59.9875,Z 153,A -154.982,B 22.2947,C -0.9475,E1 22.1719,E2 602.2851} C_DIS
LIN {X -113.5796,Y -66.6186,Z 153,A -151.9449,B 22.2955,C -0.9275,E1 22.176,E2 599.2826} C_DIS
LIN {X -112.0714,Y -69.1264,Z 153,A -150.1035,B 22.2947,C -0.9487,E1 22.1787,E2 597.3743} C_DIS
LIN {X -110.2774,Y -71.9537,Z 153,A -149.1573,B 22.2957,C -0.9228,E1 22.1801,E2 596.4913} C_DIS
LIN {X -107.5891,Y -75.914,Z 153,A -146.7717,B 22.2954,C -0.9306,E1 22.1839,E2 594.0717} C_DIS
LIN {X -104.8826,Y -79.6123,Z 153,A -144.7516,B 22.2956,C -0.9269,E1 22.1873,E2 592.0505} C_DIS
LIN {X -102.3752,Y -82.8112,Z 153,A -142.9856,B 22.2957,C -0.9225,E1 22.1903,E2 590.2865} C_DIS
LIN {X -99.5188,Y -86.2236,Z 153,A -141.0121,B 22.2959,C -0.9197,E1 22.1939,E2 588.3104} C_DIS
LIN {X -96.5675,Y -89.5162,Z 153,A -139.0886,B 22.296,C -0.9153,E1 22.1975,E2 586.3887} C_DIS
LIN {X -93.4843,Y -92.731,Z 153,A -137.1953,B 22.2963,C -0.9092,E1 22.2012,E2 584.5025} C_DIS
LIN {X -90.4425,Y -95.7001,Z 153,A -135.2381,B 22.2963,C -0.9101,E1 22.2052,E2 582.5337} C_DIS
LIN {X -87.9291,Y -98.0144,Z 153,A -133.8125,B 22.2964,C -0.9044,E1 22.2081,E2 581.1166} C_DIS
LIN {X -84.7603,Y -100.7674,Z 153,A -132.064,B 22.2967,C -0.8974,E1 22.2118,E2 579.3789} C_DIS
LIN {X -81.6492,Y -103.305,Z 153,A -130.2929,B 22.2967,C -0.8952,E1 22.2157,E2 577.6061} C_DIS
LIN {X -78.4513,Y -105.7534,Z 153,A -128.3823,B 22.2967,C -0.8991,E1 22.22,E2 575.6773} C_DIS
LIN {X -74.6071,Y -108.4995,Z 153,A -126.3947,B 22.2969,C -0.8927,E1 22.2245,E2 573.699} C_DIS
LIN {X -70.8015,Y -111.0205,Z 153,A -124.2741,B 22.2968,C -0.8955,E1 22.2295,E2 571.5631} C_DIS
LIN {X -66.4992,Y -113.6497,Z 153,A -122.1967,B 22.2971,C -0.8871,E1 22.2344,E2 569.5008} C_DIS
LIN {X -62.6543,Y -115.8142,Z 153,A -120.2372,B 22.2971,C -0.8862,E1 22.2392,E2 567.5373} C_DIS
LIN {X -58.7419,Y -117.8453,Z 153,A -118.5573,B 22.2976,C -0.8731,E1 22.2433,E2 565.8869} C_DIS
LIN {X -56.623,Y -118.8768,Z 153,A -117.3864,B 22.2974,C -0.8784,E1 22.2463,E2 564.6986} C_DIS
LIN {X -52.9433,Y -120.5629,Z 153,A -115.4051,B 22.2971,C -0.8863,E1 22.2515,E2 562.6908} C_DIS
LIN {X -49.1427,Y -122.1591,Z 153,A -113.8161,B 22.2976,C -0.8753,E1 22.2555,E2 561.1271} C_DIS
LIN {X -45.9568,Y -123.3932,Z 153,A -112.323,B 22.2976,C -0.8741,E1 22.2594,E2 559.6334} C_DIS
LIN {X -42.5472,Y -124.6113,Z 153,A -110.7983,B 22.2977,C -0.8705,E1 22.2634,E2 558.1151} C_DIS
LIN {X -37.0477,Y -126.3541,Z 153,A -108.5734,B 22.2983,C -0.8556,E1 22.2693,E2 555.925} C_DIS
LIN {X -32.5597,Y -127.5844,Z 153,A -106.26,B 22.2978,C -0.8674,E1 22.2756,E2 553.5764} C_DIS
LIN {X -29.4028,Y -128.3487,Z 153,A -104.888,B 22.2979,C -0.8648,E1 22.2793,E2 552.2094} C_DIS
LIN {X -26.2096,Y -129.0386,Z 153,A -103.3914,B 22.2979,C -0.8676,E1 22.2834,E2 550.7033} C_DIS
LIN {X -22.4864,Y -129.7413,Z 153,A -101.5505,B 22.2975,C -0.8758,E1 22.2885,E2 548.8386} C_DIS
LIN {X -18.8873,Y -130.3122,Z 153,A -100.2744,B 22.2981,C -0.8611,E1 22.2919,E2 547.6} C_DIS
LIN {X -16.3729,Y -130.6536,Z 153,A -99.0978,B 22.298,C -0.8642,E1 22.2952,E2 546.4143} C_DIS
LIN {X -12.7193,Y -131.058,Z 153,A -97.4465,B 22.2979,C -0.8664,E1 22.2998,E2 544.7561} C_DIS
LIN {X -9.147,Y -131.3563,Z 153,A -95.7555,B 22.2977,C -0.8724,E1 22.3046,E2 543.0484} C_DIS
LIN {X -5.2229,Y -131.5702,Z 153,A -94.1826,B 22.2979,C -0.8662,E1 22.3089,E2 541.4916} C_DIS
LIN {X -1.5498,Y -131.6662,Z 153,A -92.4825,B 22.2977,C -0.8711,E1 22.3137,E2 539.7784} C_DIS
LIN {X -1.5498,Y -131.6662,Z 153,A -92.4825,B 22.2977,C -0.8711,E1 22.3137,E2 539.7784} C_DIS
Enddeposition()
LIN {X 0.9146,Y -130.7293,Z 153,A -91.255,B 21.3103,C -0.7226,E1 21.3244,E2 538.838} C_DIS
Startdeposition()
$VEL.CP = VEL_PRINT
LIN {X -3.3297,Y -130.6915,Z 153,A -93.7818,B 21.3112,C -0.6931,E1 21.3171,E2 541.4461} C_DIS
LIN {X -6.1867,Y -130.5876,Z 153,A -95.2051,B 21.3114,C -0.6857,E1 21.3131,E2 542.8902} C_DIS
LIN {X -10.7282,Y -130.2929,Z 153,A -97.0003,B 21.3112,C -0.6943,E1 21.3082,E2 544.6624} C_DIS
LIN {X -14.1676,Y -129.9636,Z 153,A -98.4693,B 21.3111,C -0.6965,E1 21.3041,E2 546.1265} C_DIS
LIN {X -16.6444,Y -129.67,Z 153,A -99.7145,B 21.3113,C -0.6901,E1 21.3006,E2 547.3901} C_DIS
LIN {X -22.5267,Y -128.7789,Z 153,A -102.2803,B 21.3113,C -0.6927,E1 21.2935,E2 549.9517} C_DIS
LIN {X -26.1139,Y -128.0987,Z 153,A -103.7758,B 21.311,C -0.6979,E1 21.2895,E2 551.435} C_DIS
LIN {X -29.3479,Y -127.3968,Z 153,A -105.1512,B 21.311,C -0.7018,E1 21.2857,E2 552.8016} C_DIS
LIN {X -32.9967,Y -126.5026,Z 153,A -107.0455,B 21.3112,C -0.6922,E1 21.2805,E2 554.7257} C_DIS
LIN {X -37.3196,Y -125.2948,Z 153,A -108.9602,B 21.3112,C -0.6957,E1 21.2754,E2 556.6342} C_DIS
LIN {X -41.0513,Y -124.121,Z 153,A -110.5887,B 21.311,C -0.7007,E1 21.2711,E2 558.2524} C_DIS
LIN {X -44.5085,Y -122.9235,Z 153,A -112.2106,B 21.311,C -0.7014,E1 21.2668,E2 559.8764} C_DIS
LIN {X -47.9303,Y -121.6314,Z 153,A -113.7499,B 21.3108,C -0.7056,E1 21.2628,E2 561.408} C_DIS
LIN {X -53.2212,Y -119.4096,Z 153,A -116.3103,B 21.3108,C -0.7063,E1 21.2563,E2 563.9733} C_DIS
LIN {X -56.7264,Y -117.7854,Z 153,A -118.211,B 21.311,C -0.6996,E1 21.2514,E2 565.8983} C_DIS
LIN {X -60.5402,Y -115.871,Z 153,A -119.918,B 21.3107,C -0.7088,E1 21.2472,E2 567.5854} C_DIS
LIN {X -64.365,Y -113.7933,Z 153,A -121.9154,B 21.3107,C -0.7077,E1 21.2423,E2 569.5928} C_DIS
LIN {X -67.0794,Y -112.2142,Z 153,A -123.8223,B 21.3114,C -0.6877,E1 21.2376,E2 571.5617} C_DIS
LIN {X -71.1808,Y -109.6582,Z 153,A -125.4195,B 21.3106,C -0.7125,E1 21.234,E2 573.0967} C_DIS
LIN {X -74.0252,Y -107.7586,Z 153,A -127.2977,B 21.311,C -0.6993,E1 21.2295,E2 575.0188} C_DIS
LIN {X -77.3257,Y -105.4153,Z 153,A -128.6698,B 21.3104,C -0.7188,E1 21.2265,E2 576.3427} C_DIS
LIN {X -80.6305,Y -102.9096,Z 153,A -130.5773,B 21.3104,C -0.7184,E1 21.2223,E2 578.2597} C_DIS
LIN {X -84.3091,Y -99.9186,Z 153,A -132.6221,B 21.3102,C -0.7236,E1 21.2179,E2 580.2994} C_DIS
LIN {X -87.7899,Y -96.874,Z 153,A -135.049,B 21.3106,C -0.7114,E1 21.2128,E2 582.7718} C_DIS
LIN {X -90.8207,Y -94.0386,Z 153,A -136.4435,B 21.3099,C -0.7323,E1 21.2101,E2 584.1152} C_DIS
LIN {X -93.5123,Y -91.3627,Z 153,A -138.1467,B 21.3099,C -0.7343,E1 21.2067,E2 585.8217} C_DIS
LIN {X -96.3857,Y -88.3259,Z 153,A -139.9877,B 21.3098,C -0.7379,E1 21.2032,E2 587.6623} C_DIS
LIN {X -99.3213,Y -85.0121,Z 153,A -141.9904,B 21.3097,C -0.7398,E1 21.1995,E2 589.6706} C_DIS
LIN {X -102.5823,Y -81.0472,Z 153,A -144.2588,B 21.3095,C -0.7443,E1 21.1955,E2 591.939} C_DIS
LIN {X -105.462,Y -77.2621,Z 153,A -146.2949,B 21.3093,C -0.7514,E1 21.1921,E2 593.9675} C_DIS
LIN {X -107.9798,Y -73.7028,Z 153,A -148.2066,B 21.3092,C -0.7561,E1 21.1891,E2 595.8772} C_DIS
LIN {X -110.152,Y -70.4143,Z 153,A -149.9808,B 21.3091,C -0.7587,E1 21.1864,E2 597.6551} C_DIS
LIN {X -112.1024,Y -67.2668,Z 153,A -151.695,B 21.3091,C -0.7592,E1 21.1839,E2 599.3783} C_DIS
LIN {X -115.4128,Y -61.4126,Z 153,A -154.6115,B 21.3087,C -0.7684,E1 21.18,E2 602.2877} C_DIS
LIN {X -117.1256,Y -58.0757,Z 153,A -156.0916,B 21.3083,C -0.7795,E1 21.1781,E2 603.7465} C_DIS
LIN {X -118.4251,Y -55.38,Z 153,A -157.5795,B 21.3085,C -0.7761,E1 21.1763,E2 605.2535} C_DIS
LIN {X -120.2565,Y -51.2829,Z 153,A -159.5835,B 21.3083,C -0.7802,E1 21.1741,E2 607.2593} C_DIS
LIN {X -121.448,Y -48.3922,Z 153,A -161.1882,B 21.3085,C -0.7749,E1 21.1724,E2 608.8896} C_DIS
LIN {X -122.7193,Y -45.0704,Z 153,A -162.9601,B 21.3086,C -0.771,E1 21.1707,E2 610.6841} C_DIS
LIN {X -124.2398,Y -40.6946,Z 153,A -164.5475,B 21.3078,C -0.7945,E1 21.1693,E2 612.2173} C_DIS
LIN {X -125.4362,Y -36.8366,Z 153,A -166.1335,B 21.3074,C -0.8071,E1 21.1681,E2 613.7792} C_DIS
LIN {X -126.2626,Y -33.8967,Z 153,A -167.5131,B 21.3073,C -0.8095,E1 21.167,E2 615.1618} C_DIS
LIN {X -127.0567,Y -30.7867,Z 153,A -168.9604,B 21.3072,C -0.8122,E1 21.166,E2 616.6118} C_DIS
LIN {X -127.764,Y -27.705,Z 153,A -170.2717,B 21.3069,C -0.8194,E1 21.1653,E2 617.9124} C_DIS
LIN {X -128.4018,Y -24.5801,Z 153,A -171.8251,B 21.3069,C -0.8175,E1 21.1644,E2 619.482} C_DIS
LIN {X -129.1036,Y -20.587,Z 153,A -173.6639,B 21.3069,C -0.8206,E1 21.1635,E2 621.3253} C_DIS
LIN {X -129.6531,Y -16.7735,Z 153,A -175.4808,B 21.3069,C -0.8208,E1 21.1629,E2 623.1546} C_DIS
LIN {X -130.079,Y -13.0779,Z 153,A -177.2536,B 21.3069,C -0.8203,E1 21.1624,E2 624.9415} C_DIS
LIN {X -130.366,Y -9.7992,Z 153,A -178.4077,B 21.3063,C -0.8362,E1 21.1621,E2 626.0597} C_DIS
LIN {X -130.564,Y -6.6558,Z 153,A 179.4741,B 21.3072,C -0.8117,E1 21.1618,E2 628.2611} C_DIS
LIN {X -130.7293,Y -1.1102,Z 153,A 177.9338,B 21.3056,C -0.8543,E1 21.1618,E2 629.6946} C_DIS
LIN {X -130.6028,Y 5.8856,Z 153,A 174.4839,B 21.3058,C -0.8489,E1 21.162,E2 633.1843} C_DIS
LIN {X -130.0777,Y 13.0918,Z 153,A 171.3956,B 21.3053,C -0.862,E1 21.1627,E2 636.2583} C_DIS
LIN {X -129.64,Y 16.8733,Z 153,A 169.8661,B 21.3049,C -0.8728,E1 21.1632,E2 637.7688} C_DIS
LIN {X -129.1549,Y 20.2558,Z 153,A 168.2894,B 21.3049,C -0.8745,E1 21.1638,E2 639.3523} C_DIS
LIN {X -128.4249,Y 24.4595,Z 153,A 166.4005,B 21.3046,C -0.8796,E1 21.1648,E2 641.2402} C_DIS
LIN {X -127.6306,Y 28.3231,Z 153,A 164.5874,B 21.3046,C -0.8817,E1 21.1658,E2 643.0603} C_DIS
LIN {X -126.7872,Y 31.8791,Z 153,A 163.0774,B 21.3042,C -0.8904,E1 21.1668,E2 644.557} C_DIS
LIN {X -125.9401,Y 35.0754,Z 153,A 161.3369,B 21.3045,C -0.8834,E1 21.1681,E2 646.3287} C_DIS
LIN {X -124.7963,Y 38.9562,Z 153,A 159.7545,B 21.304,C -0.8964,E1 21.1694,E2 647.8862} C_DIS
LIN {X -123.6208,Y 42.5341,Z 153,A 158.1305,B 21.3037,C -0.9025,E1 21.1708,E2 649.5043} C_DIS
LIN {X -122.4798,Y 45.7151,Z 153,A 156.7556,B 21.3034,C -0.9112,E1 21.1721,E2 650.8643} C_DIS
LIN {X -121.4333,Y 48.4286,Z 153,A 155.3129,B 21.3034,C -0.9084,E1 21.1736,E2 652.3244} C_DIS
LIN {X -120.0841,Y 51.6817,Z 153,A 153.8109,B 21.3032,C -0.9147,E1 21.1753,E2 653.819} C_DIS
LIN {X -118.9459,Y 54.2537,Z 153,A 152.6496,B 21.303,C -0.9211,E1 21.1766,E2 654.9701} C_DIS
LIN {X -116.9636,Y 58.4041,Z 153,A 150.2719,B 21.3033,C -0.9128,E1 21.1795,E2 657.3863} C_DIS
LIN {X -114.6707,Y 62.7878,Z 153,A 148.2713,B 21.3028,C -0.9256,E1 21.1821,E2 659.3641} C_DIS
LIN {X -112.5043,Y 66.5925,Z 153,A 146.4685,B 21.3024,C -0.9356,E1 21.1846,E2 661.1503} C_DIS
LIN {X -109.1752,Y 71.9194,Z 153,A 143.5673,B 21.3023,C -0.9374,E1 21.189,E2 664.0642} C_DIS
LIN {X -106.6059,Y 75.6768,Z 153,A 141.5233,B 21.3021,C -0.9408,E1 21.1923,E2 666.1108} C_DIS
LIN {X -104.0123,Y 79.2032,Z 153,A 139.6031,B 21.3019,C -0.9458,E1 21.1955,E2 668.0281} C_DIS
LIN {X -101.2784,Y 82.6699,Z 153,A 137.6975,B 21.3017,C -0.952,E1 21.1988,E2 669.9273} C_DIS
LIN {X -98.5256,Y 85.9322,Z 153,A 135.8312,B 21.3015,C -0.9569,E1 21.2022,E2 671.7902} C_DIS
LIN {X -95.6188,Y 89.1554,Z 153,A 133.883,B 21.3013,C -0.9597,E1 21.2059,E2 673.7408} C_DIS
LIN {X -92.5912,Y 92.296,Z 153,A 132.0099,B 21.3011,C -0.9658,E1 21.2095,E2 675.6066} C_DIS
LIN {X -89.6952,Y 95.1126,Z 153,A 130.2174,B 21.3009,C -0.969,E1 21.2131,E2 677.3991} C_DIS
LIN {X -86.6256,Y 97.9165,Z 153,A 128.3499,B 21.3009,C -0.9713,E1 21.217,E2 679.2692} C_DIS
LIN {X -83.2257,Y 100.8224,Z 153,A 126.3778,B 21.3007,C -0.9751,E1 21.2212,E2 681.24} C_DIS
LIN {X -79.771,Y 103.5779,Z 153,A 124.3939,B 21.3006,C -0.9772,E1 21.2256,E2 683.2266} C_DIS
LIN {X -76.1685,Y 106.2545,Z 153,A 122.4631,B 21.3003,C -0.9826,E1 21.2299,E2 685.1506} C_DIS
LIN {X -73.8122,Y 107.9047,Z 153,A 120.6899,B 21.3011,C -0.9644,E1 21.2342,E2 686.9812} C_DIS
LIN {X -69.8859,Y 110.488,Z 153,A 119.1281,B 21.3001,C -0.9883,E1 21.2377,E2 688.4831} C_DIS
LIN {X -66.0733,Y 112.8095,Z 153,A 117.1913,B 21.2999,C -0.9926,E1 21.2423,E2 690.4152} C_DIS
LIN {X -63.0186,Y 114.5444,Z 153,A 115.5871,B 21.2999,C -0.9926,E1 21.2462,E2 692.0251} C_DIS
LIN {X -59.5191,Y 116.3987,Z 153,A 113.9893,B 21.2995,C -1.001,E1 21.2501,E2 693.6048} C_DIS
LIN {X -56.3997,Y 117.9415,Z 153,A 112.4744,B 21.2994,C -1.0037,E1 21.2539,E2 695.1166} C_DIS
LIN {X -53.7728,Y 119.1629,Z 153,A 110.7068,B 21.3002,C -0.9853,E1 21.2586,E2 696.9404} C_DIS
LIN {X -50.1576,Y 120.7287,Z 153,A 109.0843,B 21.2999,C -0.9919,E1 21.2627,E2 698.5491} C_DIS
LIN {X -46.9496,Y 122.0126,Z 153,A 107.7727,B 21.2995,C -1.0021,E1 21.2661,E2 699.8358} C_DIS
LIN {X -43.0137,Y 123.4545,Z 153,A 106.0319,B 21.2992,C -1.0083,E1 21.2706,E2 701.5635} C_DIS
LIN {X -39.3942,Y 124.6572,Z 153,A 104.32,B 21.2992,C -1.0086,E1 21.2752,E2 703.2784} C_DIS
LIN {X -35.3646,Y 125.8592,Z 153,A 102.4707,B 21.2992,C -1.0102,E1 21.2801,E2 705.1268} C_DIS
LIN {X -27.4933,Y 127.8097,Z 153,A 98.6403,B 21.2995,C -1.0019,E1 21.2906,E2 708.9862} C_DIS
LIN {X -24.1578,Y 128.4821,Z 153,A 97.0546,B 21.2996,C -0.9991,E1 21.295,E2 710.5817} C_DIS
LIN {X -20.3342,Y 129.1428,Z 153,A 95.7536,B 21.2988,C -1.0169,E1 21.2984,E2 711.8351} C_DIS
LIN {X -12.1123,Y 130.1717,Z 153,A 91.8552,B 21.2992,C -1.0076,E1 21.3093,E2 715.7621} C_DIS
LIN {X -6.814,Y 130.5561,Z 153,A 89.8097,B 21.2986,C -1.0203,E1 21.3149,E2 717.7734} C_DIS
LIN {X -3.0634,Y 130.6986,Z 153,A 87.9139,B 21.2991,C -1.0101,E1 21.3203,E2 719.6976} C_DIS
LIN {X 1.6052,Y 130.725,Z 153,A 86.2251,B 21.2984,C -1.0256,E1 21.3249,E2 721.3437} C_DIS
LIN {X 6.0574,Y 130.5941,Z 153,A 84.1002,B 21.2987,C -1.0183,E1 21.3309,E2 723.488} C_DIS
LIN {X 9.8117,Y 130.3651,Z 153,A 82.4901,B 21.2987,C -1.0199,E1 21.3354,E2 725.093} C_DIS
LIN {X 12.664,Y 130.1188,Z 153,A 81.0285,B 21.2991,C -1.0109,E1 21.3395,E2 726.5781} C_DIS
LIN {X 19.4595,Y 129.2782,Z 153,A 78.183,B 21.2988,C -1.0167,E1 21.3473,E2 729.4048} C_DIS
LIN {X 22.9,Y 128.7121,Z 153,A 76.8427,B 21.2985,C -1.0242,E1 21.3509,E2 730.7228} C_DIS
LIN {X 26.7822,Y 127.9627,Z 153,A 74.6821,B 21.2993,C -1.005,E1 21.357,E2 732.9331} C_DIS
LIN {X 30.0058,Y 127.2449,Z 153,A 73.4544,B 21.299,C -1.0136,E1 21.3603,E2 734.135} C_DIS
LIN {X 34.1533,Y 126.1942,Z 153,A 71.6574,B 21.2989,C -1.0158,E1 21.3651,E2 735.9227} C_DIS
LIN {X 38.019,Y 125.0831,Z 153,A 69.9336,B 21.2989,C -1.0162,E1 21.3697,E2 737.6419} C_DIS
LIN {X 41.5351,Y 123.9599,Z 153,A 68.2775,B 21.2989,C -1.0132,E1 21.3741,E2 739.3025} C_DIS
LIN {X 45.0375,Y 122.7327,Z 153,A 66.7205,B 21.2989,C -1.0147,E1 21.3782,E2 740.8515} C_DIS
LIN {X 50.049,Y 120.774,Z 153,A 64.3397,B 21.2991,C -1.0113,E1 21.3844,E2 743.2353} C_DIS
LIN {X 52.9331,Y 119.5385,Z 153,A 62.9747,B 21.2991,C -1.0102,E1 21.3879,E2 744.5994} C_DIS
LIN {X 56.2132,Y 118.0306,Z 153,A 61.3841,B 21.2992,C -1.0079,E1 21.3919,E2 746.1913} C_DIS
LIN {X 59.5558,Y 116.38,Z 153,A 59.7052,B 21.2994,C -1.0038,E1 21.3961,E2 747.8759} C_DIS
LIN {X 63.5078,Y 114.2735,Z 153,A 57.2309,B 21.3005,C -0.9786,E1 21.4023,E2 750.4108} C_DIS
LIN {X 67.5079,Y 111.9569,Z 153,A 55.6972,B 21.2997,C -0.9972,E1 21.4058,E2 751.8878} C_DIS
LIN {X 71.2028,Y 109.644,Z 153,A 53.9409,B 21.2995,C -1.0011,E1 21.4099,E2 753.6267} C_DIS
LIN {X 74.3641,Y 107.5256,Z 153,A 52.0946,B 21.3,C -0.9904,E1 21.4142,E2 755.495} C_DIS
LIN {X 77.9786,Y 104.9333,Z 153,A 50.1724,B 21.3,C -0.9882,E1 21.4186,E2 757.415} C_DIS
LIN {X 81.4792,Y 102.2388,Z 153,A 48.2909,B 21.3001,C -0.9871,E1 21.4227,E2 759.2912} C_DIS
LIN {X 84.8845,Y 99.43,Z 153,A 46.3238,B 21.3004,C -0.9819,E1 21.4269,E2 761.2634} C_DIS
LIN {X 87.2203,Y 97.3871,Z 153,A 44.7256,B 21.301,C -0.9685,E1 21.4303,E2 762.8906} C_DIS
LIN {X 89.7684,Y 95.0432,Z 153,A 43.3857,B 21.3007,C -0.9734,E1 21.433,E2 764.2108} C_DIS
LIN {X 93.1631,Y 91.7187,Z 153,A 41.3759,B 21.3007,C -0.9722,E1 21.437,E2 766.2137} C_DIS
LIN {X 96.2396,Y 88.4848,Z 153,A 39.4578,B 21.3009,C -0.9696,E1 21.4406,E2 768.1289} C_DIS
LIN {X 99.242,Y 85.1043,Z 153,A 37.7682,B 21.3005,C -0.9783,E1 21.4437,E2 769.7856} C_DIS
LIN {X 101.247,Y 82.7084,Z 153,A 36.0919,B 21.3013,C -0.9611,E1 21.4467,E2 771.4997} C_DIS
LIN {X 104.1046,Y 79.0825,Z 153,A 34.0787,B 21.3015,C -0.9567,E1 21.4502,E2 773.5136} C_DIS
LIN {X 106.066,Y 76.4315,Z 153,A 32.224,B 21.3024,C -0.9346,E1 21.4533,E2 775.4181} C_DIS
LIN {X 108.612,Y 72.7675,Z 153,A 30.718,B 21.3018,C -0.95,E1 21.4556,E2 776.8731} C_DIS
LIN {X 111.0493,Y 68.9905,Z 153,A 28.9927,B 21.3015,C -0.956,E1 21.4581,E2 778.5715} C_DIS
LIN {X 113.0373,Y 65.6829,Z 153,A 27.0899,B 21.3021,C -0.9419,E1 21.4608,E2 780.5013} C_DIS
LIN {X 115.2332,Y 61.7492,Z 153,A 25.1962,B 21.3021,C -0.9402,E1 21.4634,E2 782.3877} C_DIS
LIN {X 116.8667,Y 58.5996,Z 153,A 23.275,B 21.303,C -0.9192,E1 21.4659,E2 784.3543} C_DIS
LIN {X 118.461,Y 55.3022,Z 153,A 21.8771,B 21.3028,C -0.9241,E1 21.4675,E2 785.7296} C_DIS
LIN {X 120.5245,Y 50.6464,Z 153,A 19.7266,B 21.3029,C -0.9215,E1 21.4699,E2 787.8733} C_DIS
LIN {X 122.3264,Y 46.1247,Z 153,A 17.7498,B 21.3029,C -0.9225,E1 21.4719,E2 789.8342} C_DIS
LIN {X 123.4707,Y 42.9671,Z 153,A 16.3089,B 21.303,C -0.9196,E1 21.4732,E2 791.2734} C_DIS
LIN {X 124.3787,Y 40.266,Z 153,A 15.0616,B 21.3032,C -0.9159,E1 21.4743,E2 792.5222} C_DIS
LIN {X 125.2956,Y 37.317,Z 153,A 13.6683,B 21.3034,C -0.91,E1 21.4754,E2 793.9222} C_DIS
LIN {X 126.3914,Y 33.4138,Z 153,A 11.3019,B 21.3047,C -0.8776,E1 21.4772,E2 796.3611} C_DIS
LIN {X 127.5879,Y 28.5112,Z 153,A 9.7288,B 21.3038,C -0.9001,E1 21.4781,E2 797.8616} C_DIS
LIN {X 128.701,Y 22.9622,Z 153,A 7.2684,B 21.3041,C -0.8934,E1 21.4794,E2 800.3233} C_DIS
LIN {X 129.3291,Y 19.1211,Z 153,A 5.0094,B 21.3053,C -0.8625,E1 21.4804,E2 802.6507} C_DIS
LIN {X 129.9283,Y 14.4958,Z 153,A 3.236,B 21.3051,C -0.8686,E1 21.481,E2 804.3952} C_DIS
LIN {X 130.2533,Y 11.1966,Z 153,A 2.1053,B 21.3047,C -0.8789,E1 21.4812,E2 805.4897} C_DIS
LIN {X 130.5267,Y 7.38,Z 153,A 0.5311,B 21.3047,C -0.8783,E1 21.4815,E2 807.0543} C_DIS
LIN {X 130.6905,Y 3.3671,Z 153,A -1.2674,B 21.305,C -0.871,E1 21.4817,E2 808.8602} C_DIS
LIN {X 130.7306,Y 0.8447,Z 153,A -2.6692,B 21.3056,C -0.8537,E1 21.4817,E2 810.2991} C_DIS
LIN {X 130.6612,Y -4.4045,Z 153,A -4.7796,B 21.3056,C -0.8552,E1 21.4816,E2 812.3906} C_DIS
LIN {X 130.4758,Y -8.2064,Z 153,A -6.3297,B 21.3056,C -0.8553,E1 21.4813,E2 813.9293} C_DIS
LIN {X 130.1384,Y -12.4598,Z 153,A -8.5569,B 21.3064,C -0.8328,E1 21.4808,E2 816.2022} C_DIS
LIN {X 129.728,Y -16.1975,Z 153,A -9.9429,B 21.3062,C -0.8397,E1 21.4803,E2 817.5597} C_DIS
LIN {X 129.261,Y -19.5702,Z 153,A -12.0007,B 21.3073,C -0.8088,E1 21.4795,E2 819.6874} C_DIS
LIN {X 128.3619,Y -24.789,Z 153,A -13.6225,B 21.3064,C -0.8338,E1 21.4787,E2 821.2297} C_DIS
LIN {X 127.0407,Y -30.8528,Z 153,A -16.3223,B 21.3067,C -0.8261,E1 21.477,E2 823.9317} C_DIS
LIN {X 125.6009,Y -36.274,Z 153,A -19.1378,B 21.3076,C -0.8019,E1 21.4749,E2 826.7941} C_DIS
LIN {X 124.526,Y -39.805,Z 153,A -20.407,B 21.3072,C -0.813,E1 21.4738,E2 828.0243} C_DIS
LIN {X 123.1096,Y -43.9923,Z 153,A -22.241,B 21.3072,C -0.8119,E1 21.4722,E2 829.8491} C_DIS
LIN {X 122.2149,Y -46.4223,Z 153,A -24.5611,B 21.3092,C -0.7539,E1 21.4697,E2 832.3123} C_DIS
LIN {X 119.2865,Y -53.4965,Z 153,A -26.6536,B 21.3076,C -0.8018,E1 21.4675,E2 834.2602} C_DIS
LIN {X 115.1655,Y -61.8753,Z 153,A -30.8196,B 21.3081,C -0.7863,E1 21.4623,E2 838.4421} C_DIS
LIN {X 113.2507,Y -65.3144,Z 153,A -32.6059,B 21.3084,C -0.7785,E1 21.4598,E2 840.2387} C_DIS
LIN {X 111.0119,Y -69.0506,Z 153,A -34.4606,B 21.3084,C -0.7756,E1 21.4571,E2 842.09} C_DIS
LIN {X 108.6095,Y -72.7713,Z 153,A -36.4159,B 21.3087,C -0.7696,E1 21.4541,E2 844.0501} C_DIS
LIN {X 106.1092,Y -76.3717,Z 153,A -38.2152,B 21.3087,C -0.77,E1 21.4512,E2 845.8378} C_DIS
LIN {X 104.1636,Y -79.0043,Z 153,A -39.8531,B 21.3091,C -0.7568,E1 21.4485,E2 847.5024} C_DIS
LIN {X 101.0131,Y -82.9946,Z 153,A -41.7011,B 21.3087,C -0.7685,E1 21.4453,E2 849.3082} C_DIS
LIN {X 97.4703,Y -87.1274,Z 153,A -44.1533,B 21.309,C -0.7593,E1 21.4408,E2 851.7722} C_DIS
LIN {X 93.5241,Y -91.3506,Z 153,A -46.7818,B 21.3094,C -0.7487,E1 21.4357,E2 854.4161} C_DIS
LIN {X 88.5515,Y -96.1784,Z 153,A -49.6834,B 21.3094,C -0.7478,E1 21.4299,E2 857.3058} C_DIS
LIN {X 84.9327,Y -99.389,Z 153,A -52.0117,B 21.3099,C -0.7335,E1 21.425,E2 859.6624} C_DIS
LIN {X 82.4921,Y -101.4238,Z 153,A -53.6639,B 21.3104,C -0.7187,E1 21.4213,E2 861.3476} C_DIS
LIN {X 79.6359,Y -103.6805,Z 153,A -54.9049,B 21.31,C -0.7314,E1 21.4187,E2 862.5483} C_DIS
LIN {X 76.383,Y -106.1011,Z 153,A -56.712,B 21.3101,C -0.7264,E1 21.4146,E2 864.3615} C_DIS
LIN {X 72.8908,Y -108.5297,Z 153,A -58.5983,B 21.3103,C -0.7217,E1 21.4102,E2 866.2529} C_DIS
LIN {X 69.2742,Y -110.8728,Z 153,A -60.463,B 21.3103,C -0.7192,E1 21.4058,E2 868.1171} C_DIS
LIN {X 65.5084,Y -113.1383,Z 153,A -62.3793,B 21.3105,C -0.7162,E1 21.4012,E2 870.0347} C_DIS
LIN {X 61.6489,Y -115.2871,Z 153,A -64.2091,B 21.3105,C -0.7177,E1 21.3968,E2 871.8541} C_DIS
LIN {X 55.2598,Y -118.4807,Z 153,A -67.3579,B 21.3106,C -0.7119,E1 21.3889,E2 875.0087} C_DIS
LIN {X 52.0547,Y -119.9228,Z 153,A -68.7355,B 21.3104,C -0.717,E1 21.3854,E2 876.3684} C_DIS
LIN {X 46.7221,Y -122.1011,Z 153,A -71.4462,B 21.3108,C -0.7051,E1 21.3783,E2 879.1043} C_DIS
LIN {X 43.2265,Y -123.3807,Z 153,A -73.0868,B 21.3108,C -0.7026,E1 21.374,E2 880.7477} C_DIS
LIN {X 39.4409,Y -124.6423,Z 153,A -75.9942,B 21.3125,C -0.6497,E1 21.3659,E2 883.7942} C_DIS
LIN {X 31.6675,Y -126.8409,Z 153,A -78.0794,B 21.3107,C -0.71,E1 21.3607,E2 885.7098} C_DIS
LIN {X 24.155,Y -128.4831,Z 153,A -81.6352,B 21.311,C -0.6988,E1 21.3509,E2 889.2909} C_DIS
LIN {X 18.0003,Y -129.4892,Z 153,A -84.4943,B 21.3112,C -0.6913,E1 21.343,E2 892.1672} C_DIS
LIN {X 14.0455,Y -129.9768,Z 153,A -86.0172,B 21.311,C -0.7001,E1 21.3388,E2 893.6645} C_DIS
LIN {X 8.7824,Y -130.4403,Z 153,A -88.5517,B 21.3113,C -0.6895,E1 21.3317,E2 896.2268} C_DIS
LIN {X 4.8717,Y -130.643,Z 153,A -90.1934,B 21.3113,C -0.6921,E1 21.3271,E2 897.8605} C_DIS
LIN {X 0.9146,Y -130.7293,Z 153,A -91.2514,B 21.3103,C -0.7213,E1 21.3244,E2 898.838} C_DIS
Enddeposition()
LIN {X 0.9146,Y -130.7293,Z 153,A -91.2514,B 21.3103,C -0.7213,E1 21.3244,E2 898.838} C_DIS
Startdeposition()
$VEL.CP = VEL_PRINT
LIN {X 2.6508,Y -129.7673,Z 153,A -89.9791,B 20.1281,C -0.5693,E1 20.141,E2 897.8697} C_DIS
LIN {X 6.8095,Y -129.6149,Z 153,A -88.2656,B 20.1282,C -0.5648,E1 20.1457,E2 896.17} C_DIS
LIN {X 11.566,Y -129.2785,Z 153,A -85.8323,B 20.1278,C -0.5794,E1 20.1526,E2 893.6959} C_DIS
LIN {X 14.8495,Y -128.9421,Z 153,A -84.8276,B 20.1283,C -0.5613,E1 20.1552,E2 892.7445} C_DIS
LIN {X 23.872,Y -127.58,Z 153,A -80.6745,B 20.1281,C -0.5692,E1 20.1668,E2 888.5738} C_DIS
LIN {X 30.6949,Y -126.1116,Z 153,A -77.6437,B 20.1281,C -0.5697,E1 20.175,E2 885.5465} C_DIS
LIN {X 34.13,Y -125.2273,Z 153,A -75.4888,B 20.1274,C -0.5962,E1 20.181,E2 883.3192} C_DIS
LIN {X 38.4005,Y -123.9831,Z 153,A -74.088,B 20.128,C -0.5745,E1 20.1846,E2 881.9847} C_DIS
LIN {X 42.5862,Y -122.6076,Z 153,A -72.1443,B 20.128,C -0.5768,E1 20.1897,E2 880.0392} C_DIS
LIN {X 45.7589,Y -121.4594,Z 153,A -70.6398,B 20.1278,C -0.5793,E1 20.1937,E2 878.5314} C_DIS
LIN {X 53.329,Y -118.3315,Z 153,A -67.5361,B 20.1283,C -0.5625,E1 20.2015,E2 875.4855} C_DIS
LIN {X 59.8222,Y -115.186,Z 153,A -63.8533,B 20.1276,C -0.5885,E1 20.2109,E2 871.7399} C_DIS
LIN {X 63.4374,Y -113.2361,Z 153,A -61.984,B 20.1274,C -0.594,E1 20.2155,E2 869.8617} C_DIS
LIN {X 66.9468,Y -111.1975,Z 153,A -60.2213,B 20.1274,C -0.5959,E1 20.2197,E2 868.1003} C_DIS
LIN {X 70.5859,Y -108.9235,Z 153,A -58.3843,B 20.1274,C -0.5969,E1 20.224,E2 866.2679} C_DIS
LIN {X 73.887,Y -106.7121,Z 153,A -56.5827,B 20.1272,C -0.6024,E1 20.2282,E2 864.4583} C_DIS
LIN {X 77.3189,Y -104.2522,Z 153,A -54.1897,B 20.1264,C -0.6291,E1 20.2338,E2 861.9987} C_DIS
LIN {X 81.1907,Y -101.2665,Z 153,A -52.6354,B 20.127,C -0.6074,E1 20.237,E2 860.5147} C_DIS
LIN {X 84.3745,Y -98.6294,Z 153,A -50.7271,B 20.1268,C -0.6149,E1 20.2411,E2 858.5939} C_DIS
LIN {X 88.6216,Y -94.8311,Z 153,A -48.0096,B 20.1264,C -0.6295,E1 20.2468,E2 855.8484} C_DIS
LIN {X 91.1088,Y -92.4444,Z 153,A -46.767,B 20.1267,C -0.6208,E1 20.2492,E2 854.6373} C_DIS
LIN {X 93.9997,Y -89.5031,Z 153,A -44.9256,B 20.1265,C -0.6261,E1 20.2528,E2 852.7908} C_DIS
LIN {X 97.4351,Y -85.7506,Z 153,A -42.5071,B 20.1261,C -0.6392,E1 20.2573,E2 850.3481} C_DIS
LIN {X 100.5715,Y -82.0491,Z 153,A -40.5958,B 20.1262,C -0.6346,E1 20.2607,E2 848.4614} C_DIS
LIN {X 103.3427,Y -78.5309,Z 153,A -38.4885,B 20.1259,C -0.6454,E1 20.2643,E2 846.3355} C_DIS
LIN {X 105.3986,Y -75.749,Z 153,A -37.0761,B 20.1259,C -0.6444,E1 20.2666,E2 844.9346} C_DIS
LIN {X 107.8447,Y -72.2235,Z 153,A -35.1947,B 20.1259,C -0.649,E1 20.2695,E2 843.0518} C_DIS
LIN {X 110.157,Y -68.645,Z 153,A -33.3409,B 20.1257,C -0.653,E1 20.2723,E2 841.1983} C_DIS
LIN {X 112.4552,Y -64.8118,Z 153,A -31.4077,B 20.1256,C -0.6568,E1 20.2751,E2 839.2668} C_DIS
LIN {X 114.4377,Y -61.2433,Z 153,A -28.7503,B 20.1242,C -0.7,E1 20.2787,E2 836.5026} C_DIS
LIN {X 117.3476,Y -55.4618,Z 153,A -26.8825,B 20.1253,C -0.6643,E1 20.2808,E2 834.7504} C_DIS
LIN {X 118.5593,Y -52.8196,Z 153,A -25.5562,B 20.1251,C -0.67,E1 20.2823,E2 833.4169} C_DIS
LIN {X 121.0792,Y -46.7559,Z 153,A -22.7176,B 20.125,C -0.6759,E1 20.2853,E2 830.581} C_DIS
LIN {X 122.1241,Y -43.9536,Z 153,A -21.4288,B 20.1249,C -0.6786,E1 20.2866,E2 829.2938} C_DIS
LIN {X 123.249,Y -40.6942,Z 153,A -19.8656,B 20.1247,C -0.685,E1 20.288,E2 827.7232} C_DIS
LIN {X 125.1559,Y -34.3885,Z 153,A -17.0296,B 20.1245,C -0.6907,E1 20.2902,E2 824.8914} C_DIS
LIN {X 125.9217,Y -31.4673,Z 153,A -15.552,B 20.1241,C -0.7012,E1 20.2912,E2 823.3942} C_DIS
LIN {X 127.3131,Y -25.2595,Z 153,A -12.9188,B 20.1241,C -0.7022,E1 20.2928,E2 820.7776} C_DIS
LIN {X 128.3655,Y -19.2095,Z 153,A -10.2409,B 20.1239,C -0.7092,E1 20.294,E2 818.0994} C_DIS
LIN {X 129.2408,Y -11.9709,Z 153,A -6.626,B 20.1229,C -0.7369,E1 20.2951,E2 814.4318} C_DIS
LIN {X 129.5257,Y -8.3391,Z 153,A -5.5349,B 20.1235,C -0.719,E1 20.2953,E2 813.4005} C_DIS
LIN {X 129.6928,Y -5.1099,Z 153,A -3.9797,B 20.1232,C -0.7292,E1 20.2955,E2 811.8277} C_DIS
LIN {X 129.7883,Y 1.267,Z 153,A -1.2512,B 20.123,C -0.7342,E1 20.2956,E2 809.1054} C_DIS
LIN {X 129.5617,Y 7.7547,Z 153,A 1.3947,B 20.123,C -0.7335,E1 20.2953,E2 806.4816} C_DIS
LIN {X 128.9199,Y 15.0356,Z 153,A 5.6124,B 20.1211,C -0.7874,E1 20.2941,E2 802.1399} C_DIS
LIN {X 128.1375,Y 20.6733,Z 153,A 7.2629,B 20.1222,C -0.7569,E1 20.2935,E2 800.5898} C_DIS
LIN {X 126.898,Y 27.2611,Z 153,A 10.338,B 20.1217,C -0.771,E1 20.2918,E2 797.4967} C_DIS
LIN {X 125.6239,Y 32.6405,Z 153,A 12.663,B 20.1216,C -0.7733,E1 20.2903,E2 795.1823} C_DIS
LIN {X 124.8586,Y 35.4518,Z 153,A 14.0801,B 20.1212,C -0.7829,E1 20.2892,E2 793.7477} C_DIS
LIN {X 123.5743,Y 39.6946,Z 153,A 15.8683,B 20.1212,C -0.7813,E1 20.2877,E2 791.9771} C_DIS
LIN {X 122.5681,Y 42.7001,Z 153,A 17.2747,B 20.1212,C -0.7857,E1 20.2864,E2 790.568} C_DIS
LIN {X 121.3762,Y 45.9811,Z 153,A 18.917,B 20.1208,C -0.7946,E1 20.2848,E2 788.9117} C_DIS
LIN {X 119.7951,Y 49.9532,Z 153,A 20.7352,B 20.1208,C -0.797,E1 20.2829,E2 787.0995} C_DIS
LIN {X 118.3657,Y 53.2525,Z 153,A 23.0371,B 20.1193,C -0.8328,E1 20.2802,E2 784.7098} C_DIS
LIN {X 115.9415,Y 58.3448,Z 153,A 24.6516,B 20.1205,C -0.8013,E1 20.2783,E2 783.1975} C_DIS
LIN {X 114.7345,Y 60.6821,Z 153,A 25.895,B 20.1203,C -0.808,E1 20.2767,E2 781.943} C_DIS
LIN {X 112.8661,Y 64.0936,Z 153,A 27.6155,B 20.1201,C -0.8127,E1 20.2743,E2 780.2202} C_DIS
LIN {X 110.7538,Y 67.6777,Z 153,A 29.3937,B 20.1201,C -0.815,E1 20.2718,E2 778.447} C_DIS
LIN {X 109.0884,Y 70.3318,Z 153,A 31.2153,B 20.1191,C -0.8376,E1 20.269,E2 776.5718} C_DIS
LIN {X 107.0186,Y 73.4415,Z 153,A 32.7803,B 20.1191,C -0.8381,E1 20.2665,E2 775.0152} C_DIS
LIN {X 105.0326,Y 76.2552,Z 153,A 33.8879,B 20.1197,C -0.8239,E1 20.2648,E2 773.9553} C_DIS
LIN {X 102.8298,Y 79.2015,Z 153,A 35.6861,B 20.1192,C -0.8354,E1 20.2617,E2 772.1349} C_DIS
LIN {X 99.5312,Y 83.3082,Z 153,A 37.9206,B 20.1192,C -0.8369,E1 20.2578,E2 769.9092} C_DIS
LIN {X 96.8684,Y 86.3903,Z 153,A 39.7832,B 20.1189,C -0.8437,E1 20.2543,E2 768.0375} C_DIS
LIN {X 93.7361,Y 89.7789,Z 153,A 41.7513,B 20.1189,C -0.8452,E1 20.2506,E2 766.0759} C_DIS
LIN {X 90.8009,Y 92.7464,Z 153,A 44.002,B 20.1179,C -0.8666,E1 20.246,E2 763.7753} C_DIS
LIN {X 87.8014,Y 95.5908,Z 153,A 45.3581,B 20.1186,C -0.8502,E1 20.2433,E2 762.4737} C_DIS
LIN {X 84.957,Y 98.128,Z 153,A 47.126,B 20.1183,C -0.8572,E1 20.2396,E2 760.6947} C_DIS
LIN {X 81.5674,Y 100.9626,Z 153,A 49.0062,B 20.1183,C -0.8578,E1 20.2356,E2 758.8217} C_DIS
LIN {X 78.3184,Y 103.5033,Z 153,A 50.8716,B 20.1181,C -0.863,E1 20.2314,E2 756.9499} C_DIS
LIN {X 74.5638,Y 106.2404,Z 153,A 52.8915,B 20.1181,C -0.8652,E1 20.2268,E2 754.9327} C_DIS
LIN {X 71.3121,Y 108.4494,Z 153,A 54.4889,B 20.1181,C -0.8622,E1 20.2232,E2 753.3509} C_DIS
LIN {X 68.3584,Y 110.3353,Z 153,A 56.4973,B 20.1172,C -0.884,E1 20.2183,E2 751.2872} C_DIS
LIN {X 65.0869,Y 112.2959,Z 153,A 58.0093,B 20.1174,C -0.8792,E1 20.2147,E2 749.7951} C_DIS
LIN {X 61.5414,Y 114.2776,Z 153,A 59.6407,B 20.1176,C -0.8749,E1 20.2107,E2 748.1822} C_DIS
LIN {X 57.0484,Y 116.584,Z 153,A 61.8444,B 20.1176,C -0.8767,E1 20.2052,E2 745.981} C_DIS
LIN {X 52.3519,Y 118.7685,Z 153,A 64.029,B 20.1176,C -0.8751,E1 20.1997,E2 743.808} C_DIS
LIN {X 47.2206,Y 120.8986,Z 153,A 66.6976,B 20.1171,C -0.8866,E1 20.1927,E2 741.1137} C_DIS
LIN {X 42.3044,Y 122.7053,Z 153,A 68.7921,B 20.1174,C -0.8797,E1 20.1873,E2 739.0447} C_DIS
LIN {X 39.0913,Y 123.767,Z 153,A 70.283,B 20.1174,C -0.8808,E1 20.1833,E2 737.5541} C_DIS
LIN {X 34.7551,Y 125.0534,Z 153,A 72.2982,B 20.1173,C -0.8831,E1 20.1779,E2 735.5368} C_DIS
LIN {X 31.2022,Y 125.989,Z 153,A 73.9329,B 20.1172,C -0.8846,E1 20.1735,E2 733.9008} C_DIS
LIN {X 27.2993,Y 126.8898,Z 153,A 75.8234,B 20.1169,C -0.8906,E1 20.1683,E2 731.9962} C_DIS
LIN {X 20.1871,Y 128.2141,Z 153,A 78.6782,B 20.1175,C -0.878,E1 20.1606,E2 729.1819} C_DIS
LIN {X 14.2589,Y 129.0082,Z 153,A 81.3068,B 20.1175,C -0.8782,E1 20.1533,E2 726.5555} C_DIS
LIN {X 9.7586,Y 129.4263,Z 153,A 83.3037,B 20.1175,C -0.8785,E1 20.1477,E2 724.5591} C_DIS
LIN {X 6.6601,Y 129.6224,Z 153,A 85.548,B 20.1159,C -0.9139,E1 20.1412,E2 722.2129} C_DIS
LIN {X 1.408,Y 129.7872,Z 153,A 87.104,B 20.1173,C -0.8828,E1 20.1371,E2 720.7478} C_DIS
LIN {X -4.6412,Y 129.711,Z 153,A 89.9003,B 20.1171,C -0.8872,E1 20.1293,E2 717.9382} C_DIS
LIN {X -8.1762,Y 129.5357,Z 153,A 92.0197,B 20.1161,C -0.9091,E1 20.1232,E2 715.7544} C_DIS
LIN {X -12.9727,Y 129.1446,Z 153,A 94.133,B 20.1162,C -0.9077,E1 20.1173,E2 713.6438} C_DIS
LIN {X -17.603,Y 128.5949,Z 153,A 95.7308,B 20.117,C -0.8881,E1 20.113,E2 712.1015} C_DIS
LIN {X -21.4019,Y 128.0165,Z 153,A 98.2018,B 20.1158,C -0.9179,E1 20.106,E2 709.5406} C_DIS
LIN {X -27.5334,Y 126.8392,Z 153,A 99.9497,B 20.1176,C -0.8756,E1 20.1015,E2 707.9133} C_DIS
LIN {X -32.4029,Y 125.6843,Z 153,A 102.2579,B 20.1175,C -0.8775,E1 20.0953,E2 705.5955} C_DIS
LIN {X -35.2754,Y 124.9079,Z 153,A 103.6933,B 20.1173,C -0.881,E1 20.0913,E2 704.1471} C_DIS
LIN {X -39.2165,Y 123.727,Z 153,A 105.4653,B 20.1175,C -0.8774,E1 20.0866,E2 702.3819} C_DIS
LIN {X -42.7442,Y 122.5528,Z 153,A 107.0362,B 20.1177,C -0.8727,E1 20.0825,E2 700.8208} C_DIS
LIN {X -45.8106,Y 121.44,Z 153,A 108.4781,B 20.1177,C -0.871,E1 20.0787,E2 699.3801} C_DIS
LIN {X -51.7424,Y 119.0335,Z 153,A 110.9677,B 20.1185,C -0.8542,E1 20.0724,E2 696.9324} C_DIS
LIN {X -53.9853,Y 118.0342,Z 153,A 112.5443,B 20.1177,C -0.8717,E1 20.0683,E2 695.3} C_DIS
LIN {X -57.8174,Y 116.2047,Z 153,A 114.3162,B 20.118,C -0.8649,E1 20.0638,E2 693.5421} C_DIS
LIN {X -61.5932,Y 114.2497,Z 153,A 116.1706,B 20.1182,C -0.861,E1 20.0593,E2 691.6925} C_DIS
LIN {X -64.6586,Y 112.5438,Z 153,A 117.7774,B 20.1182,C -0.8606,E1 20.0554,E2 690.0808} C_DIS
LIN {X -68.2133,Y 110.4255,Z 153,A 120.2155,B 20.1173,C -0.881,E1 20.0494,E2 687.5734} C_DIS
LIN {X -72.2748,Y 107.8105,Z 153,A 121.8356,B 20.1183,C -0.8573,E1 20.0458,E2 686.0159} C_DIS
LIN {X -75.2928,Y 105.7248,Z 153,A 123.4627,B 20.1184,C -0.8544,E1 20.0421,E2 684.3901} C_DIS
LIN {X -78.6629,Y 103.2419,Z 153,A 125.2936,B 20.1186,C -0.8501,E1 20.038,E2 682.5636} C_DIS
LIN {X -81.8542,Y 100.7309,Z 153,A 127.155,B 20.1186,C -0.849,E1 20.0339,E2 680.6966} C_DIS
LIN {X -85.3779,Y 97.7614,Z 153,A 129.1474,B 20.1189,C -0.843,E1 20.0297,E2 678.7117} C_DIS
LIN {X -88.6938,Y 94.7639,Z 153,A 131.1337,B 20.1191,C -0.8391,E1 20.0256,E2 676.7267} C_DIS
LIN {X -91.6932,Y 91.8647,Z 153,A 132.9923,B 20.1192,C -0.8355,E1 20.0219,E2 674.8687} C_DIS
LIN {X -94.7154,Y 88.7459,Z 153,A 134.9689,B 20.1192,C -0.8331,E1 20.0181,E2 672.888} C_DIS
LIN {X -97.7441,Y 85.3978,Z 153,A 136.9322,B 20.1195,C -0.8271,E1 20.0145,E2 670.931} C_DIS
LIN {X -100.6914,Y 81.9025,Z 153,A 138.9655,B 20.1197,C -0.8226,E1 20.0109,E2 668.899} C_DIS
LIN {X -103.3887,Y 78.4703,Z 153,A 140.9427,B 20.1198,C -0.8195,E1 20.0075,E2 666.9188} C_DIS
LIN {X -106.0785,Y 74.7933,Z 153,A 142.9251,B 20.1201,C -0.8131,E1 20.0043,E2 664.9428} C_DIS
LIN {X -108.5903,Y 71.0982,Z 153,A 145.3938,B 20.1196,C -0.8265,E1 20.0004,E2 662.4193} C_DIS
LIN {X -111.0024,Y 67.2685,Z 153,A 147.0415,B 20.1203,C -0.8078,E1 19.9981,E2 660.8156} C_DIS
LIN {X -113.2198,Y 63.4664,Z 153,A 149.3735,B 20.1199,C -0.817,E1 19.9948,E2 658.4412} C_DIS
LIN {X -115.3914,Y 59.4254,Z 153,A 151.3016,B 20.1203,C -0.8075,E1 19.9923,E2 656.5276} C_DIS
LIN {X -117.1534,Y 55.8684,Z 153,A 152.6527,B 20.1211,C -0.7874,E1 19.9908,E2 655.2261} C_DIS
LIN {X -118.5322,Y 52.8803,Z 153,A 154.0814,B 20.1213,C -0.7822,E1 19.9891,E2 653.8025} C_DIS
LIN {X -119.8812,Y 49.7471,Z 153,A 155.5819,B 20.1214,C -0.7776,E1 19.9875,E2 652.3051} C_DIS
LIN {X -121.0618,Y 46.8005,Z 153,A 156.9808,B 20.1216,C -0.7733,E1 19.9861,E2 650.9087} C_DIS
LIN {X -122.2071,Y 43.7234,Z 153,A 158.4624,B 20.1217,C -0.7701,E1 19.9847,E2 649.4257} C_DIS
LIN {X -123.4841,Y 39.977,Z 153,A 160.5843,B 20.1214,C -0.7788,E1 19.9828,E2 647.263} C_DIS
LIN {X -124.5128,Y 36.644,Z 153,A 161.8362,B 20.122,C -0.7634,E1 19.9818,E2 646.0471} C_DIS
LIN {X -125.454,Y 33.2801,Z 153,A 163.3011,B 20.1222,C -0.7558,E1 19.9807,E2 644.5936} C_DIS
LIN {X -126.1649,Y 30.4741,Z 153,A 164.6238,B 20.1223,C -0.7535,E1 19.9799,E2 643.2677} C_DIS
LIN {X -126.996,Y 26.8074,Z 153,A 166.412,B 20.1223,C -0.7531,E1 19.9788,E2 641.4673} C_DIS
LIN {X -127.7857,Y 22.7397,Z 153,A 168.1361,B 20.1227,C -0.7435,E1 19.9779,E2 639.7583} C_DIS
LIN {X -128.3935,Y 19.0217,Z 153,A 169.9049,B 20.1227,C -0.7422,E1 19.9772,E2 637.9799} C_DIS
LIN {X -128.9214,Y 15.0228,Z 153,A 171.586,B 20.123,C -0.7329,E1 19.9766,E2 636.3131} C_DIS
LIN {X -129.5862,Y 7.3571,Z 153,A 174.8855,B 20.1235,C -0.7185,E1 19.9759,E2 633.0304} C_DIS
LIN {X -129.7907,Y 0.7958,Z 153,A 177.6678,B 20.124,C -0.7051,E1 19.9756,E2 630.2661} C_DIS
LIN {X -129.6776,Y -5.4991,Z 153,A -179.4811,B 20.1242,C -0.699,E1 19.9758,E2 627.411} C_DIS
LIN {X -129.404,Y -10.0648,Z 153,A -177.259,B 20.1242,C -0.7002,E1 19.9762,E2 625.1683} C_DIS
LIN {X -129.031,Y -14.0471,Z 153,A -175.1006,B 20.1238,C -0.7094,E1 19.9768,E2 622.9665} C_DIS
LIN {X -128.6062,Y -17.5261,Z 153,A -173.9267,B 20.1245,C -0.6907,E1 19.9772,E2 621.8386} C_DIS
LIN {X -128.166,Y -20.498,Z 153,A -172.4785,B 20.1245,C -0.6911,E1 19.9779,E2 620.378} C_DIS
LIN {X -127.5146,Y -24.214,Z 153,A -170.7992,B 20.1246,C -0.6866,E1 19.9787,E2 618.6995} C_DIS
LIN {X -126.7164,Y -28.1024,Z 153,A -169.125,B 20.1249,C -0.6783,E1 19.9797,E2 617.0369} C_DIS
LIN {X -125.8523,Y -31.7409,Z 153,A -167.427,B 20.1249,C -0.6751,E1 19.9808,E2 615.3355} C_DIS
LIN {X -125.0247,Y -34.8578,Z 153,A -165.9735,B 20.1251,C -0.672,E1 19.9819,E2 613.8805} C_DIS
Enddeposition()
END
